SPLINE
SPL {X  -153.420, Y  +337.122, Z    +0.000, E1  +333.501, E3 -322809.091}
SPL {X  -157.288, Y  +353.220, Z    +0.000, E1  +341.134, E3 -322821.136}
SPL {X  -159.049, Y  +365.172, Z    +0.000, E1  +347.392, E3 -322826.689}
SPL {X  -159.749, Y  +373.719, Z    +0.000, E1  +352.250, E3 -322829.310}
SPL {X  -159.988, Y  +381.741, Z    +0.000, E1  +357.172, E3 -322830.785}
SPL {X  -159.990, Y  +387.352, Z    +0.000, E1  +361.387, E3 -322831.487}
SPL {X  -159.990, Y  +391.188, Z    +0.000, E1  +365.082, E3 -322832.027}
SPL {X  -159.990, Y  +395.106, Z    +0.000, E1  +369.154, E3 -322832.768}
SPL {X  -159.990, Y  +400.303, Z    +0.000, E1  +374.927, E3 -322834.090}
SPL {X  -159.990, Y  +408.423, Z    +0.000, E1  +383.302, E3 -322837.169}
SPL {X  -159.990, Y  +438.418, Z    +0.000, E1  +401.067, E3 -322858.742}
SPL {X  -159.990, Y  +482.913, Z    +0.000, E1  +407.036, E3 -322918.096}
SPL {X  -159.990, Y  +489.230, Z    +0.000, E1  +407.019, E3 -322930.608}
SPL {X  -159.990, Y  +495.241, Z    +0.000, E1  +407.026, E3 -322942.487}
SPL {X  -159.990, Y  +501.001, Z    +0.000, E1  +407.020, E3 -322953.864}
SPL {X  -159.990, Y  +506.758, Z    +0.000, E1  +407.038, E3 -322965.210}
SPL {X  -159.990, Y  +512.807, Z    +0.000, E1  +407.022, E3 -322977.201}
SPL {X  -159.990, Y  +518.043, Z    +0.000, E1  +407.016, E3 -322987.578}
SPL {X  -159.990, Y  +523.058, Z    +0.000, E1  +407.015, E3 -322997.494}
SPL {X  -159.990, Y  +527.746, Z    +0.000, E1  +407.012, E3 -323006.768}
SPL {X  -159.990, Y  +533.771, Z    +0.000, E1  +407.034, E3 -323018.653}
SPL {X  -159.990, Y  +542.379, Z    +0.000, E1  +407.067, E3 -323035.622}
SPL {X  -159.990, Y  +549.846, Z    +0.000, E1  +407.016, E3 -323050.468}
SPL {X  -159.990, Y  +554.843, Z    +0.000, E1  +407.014, E3 -323060.346}
SPL {X  -159.990, Y  +560.453, Z    +0.000, E1  +407.023, E3 -323071.429}
SPL {X  -159.990, Y  +566.612, Z    +0.000, E1  +407.022, E3 -323083.611}
SPL {X  -159.990, Y  +572.901, Z    +0.000, E1  +407.028, E3 -323096.022}
SPL {X  -159.990, Y  +578.640, Z    +0.000, E1  +407.021, E3 -323107.374}
SPL {X  -159.990, Y  +583.515, Z    +0.000, E1  +407.019, E3 -323117.014}
SPL {X  -159.990, Y  +589.675, Z    +0.000, E1  +407.042, E3 -323129.152}
SPL {X  -159.990, Y  +596.627, Z    +0.000, E1  +407.034, E3 -323142.892}
SPL {X  -159.990, Y  +602.039, Z    +0.000, E1  +407.021, E3 -323153.598}
SPL {X  -159.990, Y  +607.106, Z    +0.000, E1  +407.028, E3 -323163.605}
SPL {X  -159.990, Y  +612.418, Z    +0.000, E1  +407.023, E3 -323174.117}
SPL {X  -159.990, Y  +618.496, Z    +0.000, E1  +407.049, E3 -323186.084}
SPL {X  -159.990, Y  +624.357, Z    +0.000, E1  +407.020, E3 -323197.710}
SPL {X  -159.990, Y  +629.711, Z    +0.000, E1  +407.034, E3 -323208.279}
SPL {X  -159.990, Y  +635.041, Z    +0.000, E1  +407.022, E3 -323218.823}
SPL {X  -159.990, Y  +639.998, Z    +0.000, E1  +407.027, E3 -323228.616}
SPL {X  -159.990, Y  +646.188, Z    +0.000, E1  +407.041, E3 -323240.842}
SPL {X  -159.990, Y  +652.067, Z    +0.000, E1  +407.023, E3 -323252.478}
SPL {X  -159.990, Y  +657.109, Z    +0.000, E1  +407.025, E3 -323262.456}
SPL {X  -159.990, Y  +662.651, Z    +0.000, E1  +407.027, E3 -323273.412}
SPL {X  -159.990, Y  +668.015, Z    +0.000, E1  +407.025, E3 -323284.012}
SPL {X  -159.972, Y  +673.909, Z    +0.000, E1  +407.029, E3 -323295.678}
SPL {X  -159.776, Y  +679.772, Z    +0.000, E1  +406.992, E3 -323307.479}
SPL {X  -159.384, Y  +685.411, Z    +0.000, E1  +406.921, E3 -323319.040}
SPL {X  -158.839, Y  +690.657, Z    +0.000, E1  +406.819, E3 -323329.995}
SPL {X  -157.875, Y  +697.431, Z    +0.000, E1  +406.688, E3 -323344.334}
SPL {X  -156.719, Y  +703.686, Z    +0.000, E1  +406.438, E3 -323357.943}
SPL {X  -155.778, Y  +707.970, Z    +0.000, E1  +406.262, E3 -323367.418}
SPL {X  -154.419, Y  +713.351, Z    +0.000, E1  +406.025, E3 -323379.450}
SPL {X  -152.913, Y  +718.557, Z    +0.000, E1  +405.729, E3 -323391.301}
SPL {X  -151.262, Y  +723.621, Z    +0.000, E1  +405.429, E3 -323402.968}
SPL {X  -149.964, Y  +727.247, Z    +0.000, E1  +405.152, E3 -323411.472}
SPL {X  -148.611, Y  +730.759, Z    +0.000, E1  +404.909, E3 -323419.733}
SPL {X  -142.577, Y  +744.086, Z    +0.000, E1  +400.686, E3 -323483.103}
ENDSPLINE

SPLINE
SPL {X  -152.566, Y  +719.671, Z    +0.000, E1  +387.682, E3 -323553.573}
SPL {X  -158.253, Y  +695.011, Z    +0.000, E1  +375.913, E3 -323570.245}
SPL {X  -159.486, Y  +684.192, Z    +0.000, E1  +369.965, E3 -323574.192}
SPL {X  -159.898, Y  +676.924, Z    +0.000, E1  +365.683, E3 -323575.890}
SPL {X  -159.990, Y  +671.720, Z    +0.000, E1  +362.298, E3 -323576.730}
SPL {X  -159.990, Y  +668.164, Z    +0.000, E1  +359.695, E3 -323577.145}
SPL {X  -159.990, Y  +665.062, Z    +0.000, E1  +356.961, E3 -323577.485}
SPL {X  -159.990, Y  +660.795, Z    +0.000, E1  +352.651, E3 -323578.147}
SPL {X  -159.990, Y  +654.574, Z    +0.000, E1  +345.673, E3 -323579.602}
SPL {X  -159.990, Y  +647.816, Z    +0.000, E1  +338.252, E3 -323581.854}
SPL {X  -159.990, Y  +640.751, Z    +0.000, E1  +331.747, E3 -323585.447}
SPL {X  -159.990, Y  +611.706, Z    +0.000, E1  +317.244, E3 -323608.221}
SPL {X  -159.990, Y  +571.318, Z    +0.000, E1  +312.417, E3 -323661.605}
SPL {X  -159.990, Y  +564.395, Z    +0.000, E1  +312.373, E3 -323674.963}
SPL {X  -159.990, Y  +555.871, Z    +0.000, E1  +312.389, E3 -323691.511}
SPL {X  -159.990, Y  +549.223, Z    +0.000, E1  +312.413, E3 -323704.434}
SPL {X  -159.990, Y  +542.502, Z    +0.000, E1  +312.392, E3 -323717.432}
SPL {X  -159.990, Y  +536.986, Z    +0.000, E1  +312.423, E3 -323728.152}
SPL {X  -159.990, Y  +532.938, Z    +0.000, E1  +312.415, E3 -323735.979}
SPL {X  -159.990, Y  +527.222, Z    +0.000, E1  +312.401, E3 -323747.045}
SPL {X  -159.990, Y  +520.237, Z    +0.000, E1  +312.390, E3 -323760.575}
SPL {X  -159.990, Y  +514.002, Z    +0.000, E1  +312.418, E3 -323772.710}
SPL {X  -159.990, Y  +507.203, Z    +0.000, E1  +312.383, E3 -323785.836}
ENDSPLINE

SPLINE
SPL {X  -159.990, Y  +517.758, Z    +0.000, E1  +318.109, E3 -323796.409}
ENDSPLINE

SPLINE
SPL {X  -159.990, Y  +516.975, Z    +0.000, E1  +319.588, E3 -323807.472}
SPL {X  -159.990, Y  +508.583, Z    +0.000, E1  +318.552, E3 -323821.777}
SPL {X  -159.990, Y  +502.438, Z    +0.000, E1  +317.876, E3 -323832.280}
SPL {X  -159.990, Y  +494.810, Z    +0.000, E1  +316.979, E3 -323844.696}
SPL {X  -159.990, Y  +485.551, Z    +0.000, E1  +316.053, E3 -323859.885}
SPL {X  -159.990, Y  +477.585, Z    +0.000, E1  +315.156, E3 -323871.796}
SPL {X  -159.990, Y  +470.785, Z    +0.000, E1  +314.453, E3 -323881.968}
SPL {X  -159.990, Y  +463.371, Z    +0.000, E1  +313.690, E3 -323892.693}
SPL {X  -159.990, Y  +455.469, Z    +0.000, E1  +312.807, E3 -323903.219}
SPL {X  -159.990, Y  +445.848, Z    +0.000, E1  +311.866, E3 -323916.312}
SPL {X  -159.990, Y  +436.400, Z    +0.000, E1  +311.449, E3 -323931.693}
SPL {X  -159.990, Y  +429.614, Z    +0.000, E1  +311.486, E3 -323944.484}
SPL {X  -159.990, Y  +423.677, Z    +0.000, E1  +311.471, E3 -323955.595}
SPL {X  -159.990, Y  +417.714, Z    +0.000, E1  +311.484, E3 -323966.806}
SPL {X  -159.990, Y  +412.449, Z    +0.000, E1  +311.483, E3 -323976.666}
SPL {X  -159.990, Y  +406.256, Z    +0.000, E1  +311.459, E3 -323988.233}
SPL {X  -159.990, Y  +399.971, Z    +0.000, E1  +311.480, E3 -324000.048}
SPL {X  -159.990, Y  +394.711, Z    +0.000, E1  +311.476, E3 -324009.906}
SPL {X  -159.990, Y  +387.710, Z    +0.000, E1  +311.455, E3 -324023.029}
SPL {X  -159.966, Y  +379.751, Z    +0.000, E1  +311.465, E3 -324037.993}
SPL {X  -159.734, Y  +373.449, Z    +0.000, E1  +311.528, E3 -324050.097}
SPL {X  -159.358, Y  +368.299, Z    +0.000, E1  +311.595, E3 -324060.156}
SPL {X  -158.689, Y  +362.140, Z    +0.000, E1  +311.691, E3 -324072.383}
SPL {X  -157.692, Y  +355.479, Z    +0.000, E1  +311.882, E3 -324085.942}
SPL {X  -156.759, Y  +350.510, Z    +0.000, E1  +312.069, E3 -324096.257}
SPL {X  -155.408, Y  +344.485, Z    +0.000, E1  +312.267, E3 -324108.892}
SPL {X  -153.753, Y  +338.264, Z    +0.000, E1  +312.613, E3 -324122.322}
SPL {X  -152.142, Y  +333.005, Z    +0.000, E1  +312.891, E3 -324133.795}
SPL {X  -150.309, Y  +327.691, Z    +0.000, E1  +313.264, E3 -324145.650}
SPL {X  -148.834, Y  +323.804, Z    +0.000, E1  +313.556, E3 -324154.413}
SPL {X  -147.343, Y  +320.157, Z    +0.000, E1  +313.838, E3 -324162.703}
SPL {X  -142.380, Y  +309.529, Z    +0.000, E1  +319.953, E3 -324235.464}
ENDSPLINE

SPLINE
SPL {X  -153.420, Y  +337.122, Z    +0.000, E1  +333.501, E3 -324292.962}
SPL {X  -157.288, Y  +353.220, Z    +0.000, E1  +341.134, E3 -324305.007}
SPL {X  -159.049, Y  +365.172, Z    +0.000, E1  +347.392, E3 -324310.560}
SPL {X  -159.749, Y  +373.719, Z    +0.000, E1  +352.250, E3 -324313.181}
SPL {X  -159.988, Y  +381.741, Z    +0.000, E1  +357.172, E3 -324314.656}
SPL {X  -159.990, Y  +387.352, Z    +0.000, E1  +361.387, E3 -324315.358}
SPL {X  -159.990, Y  +392.444, Z    +0.000, E1  +366.277, E3 -324316.126}
SPL {X  -159.990, Y  +398.585, Z    +0.000, E1  +372.930, E3 -324317.506}
SPL {X  -159.990, Y  +408.423, Z    +0.000, E1  +383.302, E3 -324321.040}
SPL {X  -159.990, Y  +438.418, Z    +0.000, E1  +401.067, E3 -324342.613}
SPL {X  -159.990, Y  +482.913, Z    +0.000, E1  +407.036, E3 -324401.967}
SPL {X  -159.990, Y  +489.230, Z    +0.000, E1  +407.019, E3 -324414.479}
SPL {X  -159.990, Y  +495.241, Z    +0.000, E1  +407.026, E3 -324426.358}
SPL {X  -159.990, Y  +501.001, Z    +0.000, E1  +407.020, E3 -324437.735}
SPL {X  -159.990, Y  +506.758, Z    +0.000, E1  +407.038, E3 -324449.081}
SPL {X  -159.990, Y  +512.807, Z    +0.000, E1  +407.022, E3 -324461.072}
SPL {X  -159.990, Y  +518.043, Z    +0.000, E1  +407.016, E3 -324471.449}
SPL {X  -159.990, Y  +523.058, Z    +0.000, E1  +407.015, E3 -324481.365}
SPL {X  -159.990, Y  +527.746, Z    +0.000, E1  +407.012, E3 -324490.639}
SPL {X  -159.990, Y  +533.771, Z    +0.000, E1  +407.034, E3 -324502.523}
SPL {X  -159.990, Y  +542.379, Z    +0.000, E1  +407.067, E3 -324519.493}
SPL {X  -159.990, Y  +549.846, Z    +0.000, E1  +407.016, E3 -324534.339}
SPL {X  -159.990, Y  +554.843, Z    +0.000, E1  +407.014, E3 -324544.217}
SPL {X  -159.990, Y  +560.453, Z    +0.000, E1  +407.023, E3 -324555.299}
SPL {X  -159.990, Y  +566.612, Z    +0.000, E1  +407.022, E3 -324567.482}
SPL {X  -159.990, Y  +572.901, Z    +0.000, E1  +407.028, E3 -324579.893}
SPL {X  -159.990, Y  +578.640, Z    +0.000, E1  +407.021, E3 -324591.245}
SPL {X  -159.990, Y  +583.515, Z    +0.000, E1  +407.019, E3 -324600.885}
SPL {X  -159.990, Y  +589.675, Z    +0.000, E1  +407.042, E3 -324613.023}
SPL {X  -159.990, Y  +596.627, Z    +0.000, E1  +407.034, E3 -324626.763}
SPL {X  -159.990, Y  +602.039, Z    +0.000, E1  +407.021, E3 -324637.469}
SPL {X  -159.990, Y  +607.106, Z    +0.000, E1  +407.028, E3 -324647.476}
SPL {X  -159.990, Y  +614.483, Z    +0.000, E1  +407.064, E3 -324662.009}
SPL {X  -159.990, Y  +622.758, Z    +0.000, E1  +407.049, E3 -324678.379}
SPL {X  -159.990, Y  +629.711, Z    +0.000, E1  +407.034, E3 -324692.150}
SPL {X  -159.990, Y  +635.041, Z    +0.000, E1  +407.022, E3 -324702.694}
SPL {X  -159.990, Y  +639.998, Z    +0.000, E1  +407.027, E3 -324712.487}
SPL {X  -159.990, Y  +646.188, Z    +0.000, E1  +407.041, E3 -324724.713}
SPL {X  -159.990, Y  +652.067, Z    +0.000, E1  +407.023, E3 -324736.349}
SPL {X  -159.990, Y  +657.109, Z    +0.000, E1  +407.025, E3 -324746.327}
SPL {X  -159.990, Y  +662.651, Z    +0.000, E1  +407.027, E3 -324757.283}
SPL {X  -159.990, Y  +668.015, Z    +0.000, E1  +407.025, E3 -324767.883}
SPL {X  -159.972, Y  +673.909, Z    +0.000, E1  +407.029, E3 -324779.549}
SPL {X  -159.776, Y  +679.772, Z    +0.000, E1  +406.992, E3 -324791.350}
SPL {X  -159.384, Y  +685.411, Z    +0.000, E1  +406.921, E3 -324802.911}
SPL {X  -158.839, Y  +690.657, Z    +0.000, E1  +406.819, E3 -324813.865}
SPL {X  -157.875, Y  +697.431, Z    +0.000, E1  +406.688, E3 -324828.205}
SPL {X  -156.719, Y  +703.686, Z    +0.000, E1  +406.438, E3 -324841.814}
SPL {X  -155.432, Y  +709.417, Z    +0.000, E1  +406.234, E3 -324854.458}
SPL {X  -154.084, Y  +714.570, Z    +0.000, E1  +405.932, E3 -324866.120}
SPL {X  -152.913, Y  +718.557, Z    +0.000, E1  +405.729, E3 -324875.172}
SPL {X  -151.262, Y  +723.621, Z    +0.000, E1  +405.429, E3 -324886.839}
SPL {X  -149.074, Y  +729.584, Z    +0.000, E1  +405.040, E3 -324900.767}
SPL {X  -142.546, Y  +744.145, Z    +0.000, E1  +401.000, E3 -324963.794}
ENDSPLINE

SPLINE
SPL {X  -146.166, Y  +736.557, Z    +0.000, E1  +395.148, E3 -325007.760}
SPL {X  -153.596, Y  +716.277, Z    +0.000, E1  +386.138, E3 -325041.007}
SPL {X  -158.253, Y  +695.011, Z    +0.000, E1  +375.913, E3 -325054.116}
SPL {X  -159.486, Y  +684.192, Z    +0.000, E1  +369.965, E3 -325058.063}
SPL {X  -159.898, Y  +676.924, Z    +0.000, E1  +365.683, E3 -325059.761}
SPL {X  -159.990, Y  +671.720, Z    +0.000, E1  +362.298, E3 -325060.601}
SPL {X  -159.990, Y  +668.164, Z    +0.000, E1  +359.695, E3 -325061.016}
SPL {X  -159.990, Y  +663.705, Z    +0.000, E1  +355.772, E3 -325061.548}
SPL {X  -159.990, Y  +656.120, Z    +0.000, E1  +347.542, E3 -325063.089}
SPL {X  -159.990, Y  +647.816, Z    +0.000, E1  +338.252, E3 -325065.725}
SPL {X  -159.990, Y  +640.751, Z    +0.000, E1  +331.747, E3 -325069.318}
SPL {X  -159.990, Y  +611.706, Z    +0.000, E1  +317.244, E3 -325092.092}
SPL {X  -159.990, Y  +571.318, Z    +0.000, E1  +312.417, E3 -325145.476}
SPL {X  -159.990, Y  +564.395, Z    +0.000, E1  +312.373, E3 -325158.834}
SPL {X  -159.990, Y  +555.871, Z    +0.000, E1  +312.389, E3 -325175.382}
SPL {X  -159.990, Y  +549.223, Z    +0.000, E1  +312.413, E3 -325188.305}
SPL {X  -159.990, Y  +542.502, Z    +0.000, E1  +312.392, E3 -325201.303}
SPL {X  -159.990, Y  +536.986, Z    +0.000, E1  +312.423, E3 -325212.023}
SPL {X  -159.990, Y  +532.938, Z    +0.000, E1  +312.415, E3 -325219.850}
SPL {X  -159.990, Y  +527.222, Z    +0.000, E1  +312.401, E3 -325230.916}
SPL {X  -159.990, Y  +520.237, Z    +0.000, E1  +312.390, E3 -325244.446}
SPL {X  -159.990, Y  +514.002, Z    +0.000, E1  +312.418, E3 -325256.581}
SPL {X  -159.990, Y  +507.203, Z    +0.000, E1  +312.383, E3 -325269.707}
ENDSPLINE

SPLINE
SPL {X  -159.990, Y  +517.758, Z    +0.000, E1  +318.109, E3 -325280.280}
ENDSPLINE

SPLINE
SPL {X  -159.990, Y  +516.975, Z    +0.000, E1  +319.588, E3 -325291.343}
SPL {X  -159.990, Y  +508.583, Z    +0.000, E1  +318.552, E3 -325305.648}
SPL {X  -159.990, Y  +502.438, Z    +0.000, E1  +317.876, E3 -325316.151}
SPL {X  -159.990, Y  +494.810, Z    +0.000, E1  +316.979, E3 -325328.567}
SPL {X  -159.990, Y  +485.551, Z    +0.000, E1  +316.053, E3 -325343.756}
SPL {X  -159.990, Y  +477.585, Z    +0.000, E1  +315.156, E3 -325355.667}
SPL {X  -159.990, Y  +470.785, Z    +0.000, E1  +314.453, E3 -325365.839}
SPL {X  -159.990, Y  +463.371, Z    +0.000, E1  +313.690, E3 -325376.564}
SPL {X  -159.990, Y  +455.469, Z    +0.000, E1  +312.807, E3 -325387.090}
SPL {X  -159.990, Y  +445.848, Z    +0.000, E1  +311.866, E3 -325400.183}
SPL {X  -159.990, Y  +436.400, Z    +0.000, E1  +311.449, E3 -325415.564}
SPL {X  -159.990, Y  +429.614, Z    +0.000, E1  +311.486, E3 -325428.355}
SPL {X  -159.990, Y  +423.677, Z    +0.000, E1  +311.471, E3 -325439.466}
SPL {X  -159.990, Y  +417.714, Z    +0.000, E1  +311.484, E3 -325450.677}
SPL {X  -159.990, Y  +412.449, Z    +0.000, E1  +311.483, E3 -325460.537}
SPL {X  -159.990, Y  +406.256, Z    +0.000, E1  +311.459, E3 -325472.104}
SPL {X  -159.990, Y  +399.971, Z    +0.000, E1  +311.480, E3 -325483.919}
SPL {X  -159.990, Y  +392.623, Z    +0.000, E1  +311.440, E3 -325497.650}
SPL {X  -159.990, Y  +385.787, Z    +0.000, E1  +311.488, E3 -325510.557}
SPL {X  -159.966, Y  +379.751, Z    +0.000, E1  +311.465, E3 -325521.864}
SPL {X  -159.734, Y  +373.449, Z    +0.000, E1  +311.528, E3 -325533.968}
SPL {X  -159.230, Y  +366.920, Z    +0.000, E1  +311.592, E3 -325546.712}
SPL {X  -158.532, Y  +360.951, Z    +0.000, E1  +311.745, E3 -325558.686}
SPL {X  -157.692, Y  +355.479, Z    +0.000, E1  +311.882, E3 -325569.813}
SPL {X  -156.349, Y  +348.560, Z    +0.000, E1  +312.101, E3 -325584.153}
SPL {X  -154.984, Y  +342.790, Z    +0.000, E1  +312.392, E3 -325596.450}
SPL {X  -153.247, Y  +336.540, Z    +0.000, E1  +312.660, E3 -325609.885}
SPL {X  -150.765, Y  +328.959, Z    +0.000, E1  +313.136, E3 -325626.632}
SPL {X  -148.834, Y  +323.804, Z    +0.000, E1  +313.556, E3 -325638.284}
SPL {X  -147.343, Y  +320.157, Z    +0.000, E1  +313.838, E3 -325646.574}
SPL {X  -142.380, Y  +309.529, Z    +0.000, E1  +319.953, E3 -325719.335}
ENDSPLINE

SPLINE
SPL {X  -153.420, Y  +337.122, Z    +0.000, E1  +333.501, E3 -325776.833}
SPL {X  -157.288, Y  +353.220, Z    +0.000, E1  +341.134, E3 -325788.878}
SPL {X  -159.049, Y  +365.172, Z    +0.000, E1  +347.392, E3 -325794.431}
SPL {X  -159.749, Y  +373.719, Z    +0.000, E1  +352.250, E3 -325797.052}
SPL {X  -159.988, Y  +381.741, Z    +0.000, E1  +357.172, E3 -325798.527}
SPL {X  -159.990, Y  +387.352, Z    +0.000, E1  +361.387, E3 -325799.229}
SPL {X  -159.990, Y  +391.188, Z    +0.000, E1  +365.082, E3 -325799.769}
SPL {X  -159.990, Y  +395.106, Z    +0.000, E1  +369.154, E3 -325800.510}
SPL {X  -159.990, Y  +400.303, Z    +0.000, E1  +374.927, E3 -325801.832}
SPL {X  -159.990, Y  +408.423, Z    +0.000, E1  +383.302, E3 -325804.911}
SPL {X  -159.990, Y  +438.418, Z    +0.000, E1  +401.067, E3 -325826.484}
SPL {X  -159.990, Y  +482.913, Z    +0.000, E1  +407.036, E3 -325885.838}
SPL {X  -159.990, Y  +489.230, Z    +0.000, E1  +407.019, E3 -325898.350}
SPL {X  -159.990, Y  +495.241, Z    +0.000, E1  +407.026, E3 -325910.229}
SPL {X  -159.990, Y  +501.001, Z    +0.000, E1  +407.020, E3 -325921.606}
SPL {X  -159.990, Y  +506.758, Z    +0.000, E1  +407.038, E3 -325932.952}
SPL {X  -159.990, Y  +512.807, Z    +0.000, E1  +407.022, E3 -325944.943}
SPL {X  -159.990, Y  +518.043, Z    +0.000, E1  +407.016, E3 -325955.320}
SPL {X  -159.990, Y  +523.058, Z    +0.000, E1  +407.015, E3 -325965.236}
SPL {X  -159.990, Y  +527.746, Z    +0.000, E1  +407.012, E3 -325974.510}
SPL {X  -159.990, Y  +533.771, Z    +0.000, E1  +407.034, E3 -325986.394}
SPL {X  -159.990, Y  +542.379, Z    +0.000, E1  +407.067, E3 -326003.364}
SPL {X  -159.990, Y  +549.846, Z    +0.000, E1  +407.016, E3 -326018.210}
SPL {X  -159.990, Y  +554.843, Z    +0.000, E1  +407.014, E3 -326028.088}
SPL {X  -159.990, Y  +560.453, Z    +0.000, E1  +407.023, E3 -326039.170}
SPL {X  -159.990, Y  +566.612, Z    +0.000, E1  +407.022, E3 -326051.353}
SPL {X  -159.990, Y  +572.901, Z    +0.000, E1  +407.028, E3 -326063.764}
SPL {X  -159.990, Y  +578.640, Z    +0.000, E1  +407.021, E3 -326075.116}
SPL {X  -159.990, Y  +583.515, Z    +0.000, E1  +407.019, E3 -326084.756}
SPL {X  -159.990, Y  +589.675, Z    +0.000, E1  +407.042, E3 -326096.893}
SPL {X  -159.990, Y  +596.627, Z    +0.000, E1  +407.034, E3 -326110.634}
SPL {X  -159.990, Y  +602.039, Z    +0.000, E1  +407.021, E3 -326121.340}
SPL {X  -159.990, Y  +607.106, Z    +0.000, E1  +407.028, E3 -326131.347}
SPL {X  -159.990, Y  +612.418, Z    +0.000, E1  +407.023, E3 -326141.859}
SPL {X  -159.990, Y  +618.496, Z    +0.000, E1  +407.049, E3 -326153.826}
SPL {X  -159.990, Y  +624.357, Z    +0.000, E1  +407.020, E3 -326165.452}
SPL {X  -159.990, Y  +629.711, Z    +0.000, E1  +407.034, E3 -326176.021}
SPL {X  -159.990, Y  +635.041, Z    +0.000, E1  +407.022, E3 -326186.565}
SPL {X  -159.990, Y  +639.998, Z    +0.000, E1  +407.027, E3 -326196.358}
SPL {X  -159.990, Y  +646.188, Z    +0.000, E1  +407.041, E3 -326208.584}
SPL {X  -159.990, Y  +652.067, Z    +0.000, E1  +407.023, E3 -326220.220}
SPL {X  -159.990, Y  +657.109, Z    +0.000, E1  +407.025, E3 -326230.198}
SPL {X  -159.990, Y  +662.651, Z    +0.000, E1  +407.027, E3 -326241.154}
SPL {X  -159.990, Y  +668.015, Z    +0.000, E1  +407.025, E3 -326251.754}
SPL {X  -159.972, Y  +673.909, Z    +0.000, E1  +407.029, E3 -326263.420}
SPL {X  -159.776, Y  +679.772, Z    +0.000, E1  +406.992, E3 -326275.221}
SPL {X  -159.384, Y  +685.411, Z    +0.000, E1  +406.921, E3 -326286.782}
SPL {X  -158.839, Y  +690.657, Z    +0.000, E1  +406.819, E3 -326297.736}
SPL {X  -157.875, Y  +697.431, Z    +0.000, E1  +406.688, E3 -326312.076}
SPL {X  -156.719, Y  +703.686, Z    +0.000, E1  +406.438, E3 -326325.685}
SPL {X  -155.778, Y  +707.970, Z    +0.000, E1  +406.262, E3 -326335.160}
SPL {X  -154.419, Y  +713.351, Z    +0.000, E1  +406.025, E3 -326347.192}
SPL {X  -152.913, Y  +718.557, Z    +0.000, E1  +405.729, E3 -326359.043}
SPL {X  -151.262, Y  +723.621, Z    +0.000, E1  +405.429, E3 -326370.710}
SPL {X  -149.964, Y  +727.247, Z    +0.000, E1  +405.152, E3 -326379.214}
SPL {X  -148.611, Y  +730.759, Z    +0.000, E1  +404.909, E3 -326387.475}
SPL {X  -142.577, Y  +744.086, Z    +0.000, E1  +400.686, E3 -326450.844}
ENDSPLINE

SPLINE
SPL {X  -152.566, Y  +719.671, Z    +0.000, E1  +387.682, E3 -326521.315}
SPL {X  -158.253, Y  +695.011, Z    +0.000, E1  +375.913, E3 -326537.987}
SPL {X  -159.486, Y  +684.192, Z    +0.000, E1  +369.965, E3 -326541.934}
SPL {X  -159.898, Y  +676.924, Z    +0.000, E1  +365.683, E3 -326543.632}
SPL {X  -159.990, Y  +671.720, Z    +0.000, E1  +362.298, E3 -326544.472}
SPL {X  -159.990, Y  +668.164, Z    +0.000, E1  +359.695, E3 -326544.887}
SPL {X  -159.990, Y  +665.062, Z    +0.000, E1  +356.961, E3 -326545.227}
SPL {X  -159.990, Y  +660.795, Z    +0.000, E1  +352.651, E3 -326545.889}
SPL {X  -159.990, Y  +654.574, Z    +0.000, E1  +345.673, E3 -326547.344}
SPL {X  -159.990, Y  +647.816, Z    +0.000, E1  +338.252, E3 -326549.596}
SPL {X  -159.990, Y  +640.751, Z    +0.000, E1  +331.747, E3 -326553.189}
SPL {X  -159.990, Y  +611.706, Z    +0.000, E1  +317.244, E3 -326575.963}
SPL {X  -159.990, Y  +571.318, Z    +0.000, E1  +312.417, E3 -326629.347}
SPL {X  -159.990, Y  +564.395, Z    +0.000, E1  +312.373, E3 -326642.705}
SPL {X  -159.990, Y  +555.871, Z    +0.000, E1  +312.389, E3 -326659.253}
SPL {X  -159.990, Y  +549.223, Z    +0.000, E1  +312.413, E3 -326672.176}
SPL {X  -159.990, Y  +542.502, Z    +0.000, E1  +312.392, E3 -326685.174}
SPL {X  -159.990, Y  +536.986, Z    +0.000, E1  +312.423, E3 -326695.894}
SPL {X  -159.990, Y  +532.938, Z    +0.000, E1  +312.415, E3 -326703.721}
SPL {X  -159.990, Y  +527.222, Z    +0.000, E1  +312.401, E3 -326714.787}
SPL {X  -159.990, Y  +520.237, Z    +0.000, E1  +312.390, E3 -326728.317}
SPL {X  -159.990, Y  +514.002, Z    +0.000, E1  +312.418, E3 -326740.452}
SPL {X  -159.990, Y  +507.203, Z    +0.000, E1  +312.383, E3 -326753.578}
ENDSPLINE

SPLINE
SPL {X  -159.990, Y  +517.758, Z    +0.000, E1  +318.109, E3 -326764.151}
ENDSPLINE

SPLINE
SPL {X  -159.990, Y  +516.975, Z    +0.000, E1  +319.588, E3 -326775.214}
SPL {X  -159.990, Y  +508.583, Z    +0.000, E1  +318.552, E3 -326789.519}
SPL {X  -159.990, Y  +502.438, Z    +0.000, E1  +317.876, E3 -326800.022}
SPL {X  -159.990, Y  +494.810, Z    +0.000, E1  +316.979, E3 -326812.438}
SPL {X  -159.990, Y  +485.551, Z    +0.000, E1  +316.053, E3 -326827.627}
SPL {X  -159.990, Y  +477.585, Z    +0.000, E1  +315.156, E3 -326839.538}
SPL {X  -159.990, Y  +470.785, Z    +0.000, E1  +314.453, E3 -326849.710}
SPL {X  -159.990, Y  +463.371, Z    +0.000, E1  +313.690, E3 -326860.435}
SPL {X  -159.990, Y  +455.469, Z    +0.000, E1  +312.807, E3 -326870.961}
SPL {X  -159.990, Y  +445.848, Z    +0.000, E1  +311.866, E3 -326884.054}
SPL {X  -159.990, Y  +436.400, Z    +0.000, E1  +311.449, E3 -326899.435}
SPL {X  -159.990, Y  +429.614, Z    +0.000, E1  +311.486, E3 -326912.226}
SPL {X  -159.990, Y  +423.677, Z    +0.000, E1  +311.471, E3 -326923.337}
SPL {X  -159.990, Y  +417.714, Z    +0.000, E1  +311.484, E3 -326934.547}
SPL {X  -159.990, Y  +412.449, Z    +0.000, E1  +311.483, E3 -326944.408}
SPL {X  -159.990, Y  +406.256, Z    +0.000, E1  +311.459, E3 -326955.975}
SPL {X  -159.990, Y  +399.971, Z    +0.000, E1  +311.480, E3 -326967.790}
SPL {X  -159.990, Y  +394.711, Z    +0.000, E1  +311.476, E3 -326977.648}
SPL {X  -159.990, Y  +387.710, Z    +0.000, E1  +311.455, E3 -326990.771}
SPL {X  -159.966, Y  +379.751, Z    +0.000, E1  +311.465, E3 -327005.735}
SPL {X  -159.734, Y  +373.449, Z    +0.000, E1  +311.528, E3 -327017.839}
SPL {X  -159.358, Y  +368.299, Z    +0.000, E1  +311.595, E3 -327027.898}
SPL {X  -158.689, Y  +362.140, Z    +0.000, E1  +311.691, E3 -327040.125}
SPL {X  -157.692, Y  +355.479, Z    +0.000, E1  +311.882, E3 -327053.684}
SPL {X  -156.759, Y  +350.510, Z    +0.000, E1  +312.069, E3 -327063.999}
SPL {X  -155.408, Y  +344.485, Z    +0.000, E1  +312.267, E3 -327076.634}
SPL {X  -153.753, Y  +338.264, Z    +0.000, E1  +312.613, E3 -327090.064}
SPL {X  -152.142, Y  +333.005, Z    +0.000, E1  +312.891, E3 -327101.537}
SPL {X  -150.309, Y  +327.691, Z    +0.000, E1  +313.264, E3 -327113.392}
SPL {X  -148.834, Y  +323.804, Z    +0.000, E1  +313.556, E3 -327122.155}
SPL {X  -147.343, Y  +320.157, Z    +0.000, E1  +313.838, E3 -327130.445}
SPL {X  -142.380, Y  +309.529, Z    +0.000, E1  +319.953, E3 -327203.206}
ENDSPLINE

SPLINE
SPL {X  -153.420, Y  +337.122, Z    +0.000, E1  +333.501, E3 -327260.704}
SPL {X  -157.288, Y  +353.220, Z    +0.000, E1  +341.134, E3 -327272.749}
SPL {X  -159.049, Y  +365.172, Z    +0.000, E1  +347.392, E3 -327278.302}
SPL {X  -159.749, Y  +373.719, Z    +0.000, E1  +352.250, E3 -327280.923}
SPL {X  -159.988, Y  +381.741, Z    +0.000, E1  +357.172, E3 -327282.398}
SPL {X  -159.990, Y  +387.352, Z    +0.000, E1  +361.387, E3 -327283.100}
SPL {X  -159.990, Y  +392.444, Z    +0.000, E1  +366.277, E3 -327283.868}
SPL {X  -159.990, Y  +398.585, Z    +0.000, E1  +372.930, E3 -327285.248}
SPL {X  -159.990, Y  +408.423, Z    +0.000, E1  +383.302, E3 -327288.782}
SPL {X  -159.990, Y  +438.418, Z    +0.000, E1  +401.067, E3 -327310.355}
SPL {X  -159.990, Y  +482.913, Z    +0.000, E1  +407.036, E3 -327369.709}
SPL {X  -159.990, Y  +489.230, Z    +0.000, E1  +407.019, E3 -327382.221}
SPL {X  -159.990, Y  +495.241, Z    +0.000, E1  +407.026, E3 -327394.100}
SPL {X  -159.990, Y  +501.001, Z    +0.000, E1  +407.020, E3 -327405.477}
SPL {X  -159.990, Y  +506.758, Z    +0.000, E1  +407.038, E3 -327416.823}
SPL {X  -159.990, Y  +512.807, Z    +0.000, E1  +407.022, E3 -327428.814}
SPL {X  -159.990, Y  +518.043, Z    +0.000, E1  +407.016, E3 -327439.191}
SPL {X  -159.990, Y  +525.485, Z    +0.000, E1  +407.063, E3 -327453.836}
SPL {X  -159.990, Y  +533.771, Z    +0.000, E1  +407.034, E3 -327470.265}
SPL {X  -159.990, Y  +540.264, Z    +0.000, E1  +407.020, E3 -327483.122}
SPL {X  -159.990, Y  +547.787, Z    +0.000, E1  +407.067, E3 -327497.923}
SPL {X  -159.990, Y  +554.843, Z    +0.000, E1  +407.014, E3 -327511.959}
SPL {X  -159.990, Y  +560.453, Z    +0.000, E1  +407.023, E3 -327523.041}
SPL {X  -159.990, Y  +566.612, Z    +0.000, E1  +407.022, E3 -327535.224}
SPL {X  -159.990, Y  +572.901, Z    +0.000, E1  +407.028, E3 -327547.635}
SPL {X  -159.990, Y  +578.640, Z    +0.000, E1  +407.021, E3 -327558.987}
SPL {X  -159.990, Y  +584.969, Z    +0.000, E1  +407.043, E3 -327571.469}
SPL {X  -159.990, Y  +591.074, Z    +0.000, E1  +407.017, E3 -327583.559}
SPL {X  -159.990, Y  +596.627, Z    +0.000, E1  +407.034, E3 -327594.505}
SPL {X  -159.990, Y  +602.039, Z    +0.000, E1  +407.021, E3 -327605.211}
SPL {X  -159.990, Y  +607.106, Z    +0.000, E1  +407.028, E3 -327615.218}
SPL {X  -159.990, Y  +612.418, Z    +0.000, E1  +407.023, E3 -327625.730}
SPL {X  -159.990, Y  +618.496, Z    +0.000, E1  +407.049, E3 -327637.697}
SPL {X  -159.990, Y  +624.357, Z    +0.000, E1  +407.020, E3 -327649.323}
SPL {X  -159.990, Y  +629.711, Z    +0.000, E1  +407.034, E3 -327659.892}
SPL {X  -159.990, Y  +635.041, Z    +0.000, E1  +407.022, E3 -327670.436}
SPL {X  -159.990, Y  +642.261, Z    +0.000, E1  +407.074, E3 -327684.637}
SPL {X  -159.990, Y  +650.752, Z    +0.000, E1  +407.046, E3 -327701.464}
SPL {X  -159.990, Y  +657.109, Z    +0.000, E1  +407.025, E3 -327714.069}
SPL {X  -159.990, Y  +662.651, Z    +0.000, E1  +407.027, E3 -327725.025}
SPL {X  -159.990, Y  +668.015, Z    +0.000, E1  +407.025, E3 -327735.625}
SPL {X  -159.972, Y  +673.909, Z    +0.000, E1  +407.029, E3 -327747.291}
SPL {X  -159.776, Y  +679.772, Z    +0.000, E1  +406.992, E3 -327759.092}
SPL {X  -159.384, Y  +685.411, Z    +0.000, E1  +406.921, E3 -327770.653}
SPL {X  -158.642, Y  +692.228, Z    +0.000, E1  +406.819, E3 -327784.869}
SPL {X  -157.651, Y  +698.760, Z    +0.000, E1  +406.609, E3 -327798.863}
SPL {X  -156.719, Y  +703.686, Z    +0.000, E1  +406.438, E3 -327809.556}
SPL {X  -155.778, Y  +707.970, Z    +0.000, E1  +406.262, E3 -327819.031}
SPL {X  -154.419, Y  +713.351, Z    +0.000, E1  +406.025, E3 -327831.062}
SPL {X  -152.913, Y  +718.557, Z    +0.000, E1  +405.729, E3 -327842.914}
SPL {X  -151.262, Y  +723.621, Z    +0.000, E1  +405.429, E3 -327854.581}
SPL {X  -149.074, Y  +729.584, Z    +0.000, E1  +405.040, E3 -327868.509}
SPL {X  -142.577, Y  +744.086, Z    +0.000, E1  +400.686, E3 -327934.715}
ENDSPLINE

SPLINE
SPL {X  -152.566, Y  +719.671, Z    +0.000, E1  +387.682, E3 -328005.186}
SPL {X  -158.253, Y  +695.011, Z    +0.000, E1  +375.913, E3 -328021.858}
SPL {X  -159.486, Y  +684.192, Z    +0.000, E1  +369.965, E3 -328025.805}
SPL {X  -159.898, Y  +676.924, Z    +0.000, E1  +365.683, E3 -328027.503}
SPL {X  -159.990, Y  +671.720, Z    +0.000, E1  +362.298, E3 -328028.343}
SPL {X  -159.990, Y  +668.164, Z    +0.000, E1  +359.695, E3 -328028.758}
SPL {X  -159.990, Y  +665.062, Z    +0.000, E1  +356.961, E3 -328029.098}
SPL {X  -159.990, Y  +660.795, Z    +0.000, E1  +352.651, E3 -328029.760}
SPL {X  -159.990, Y  +654.574, Z    +0.000, E1  +345.673, E3 -328031.215}
SPL {X  -159.990, Y  +644.002, Z    +0.000, E1  +334.724, E3 -328035.412}
SPL {X  -159.990, Y  +611.706, Z    +0.000, E1  +317.244, E3 -328059.834}
SPL {X  -159.990, Y  +571.318, Z    +0.000, E1  +312.417, E3 -328113.218}
SPL {X  -159.990, Y  +564.395, Z    +0.000, E1  +312.373, E3 -328126.576}
SPL {X  -159.990, Y  +555.871, Z    +0.000, E1  +312.389, E3 -328143.124}
SPL {X  -159.990, Y  +549.223, Z    +0.000, E1  +312.413, E3 -328156.047}
SPL {X  -159.990, Y  +542.502, Z    +0.000, E1  +312.392, E3 -328169.045}
SPL {X  -159.990, Y  +534.538, Z    +0.000, E1  +312.385, E3 -328184.449}
SPL {X  -159.990, Y  +527.222, Z    +0.000, E1  +312.401, E3 -328198.658}
SPL {X  -159.990, Y  +520.237, Z    +0.000, E1  +312.390, E3 -328212.188}
SPL {X  -159.990, Y  +512.328, Z    +0.000, E1  +312.388, E3 -328227.522}
SPL {X  -159.990, Y  +505.755, Z    +0.000, E1  +312.413, E3 -328240.299}
ENDSPLINE

SPLINE
SPL {X  -159.990, Y  +518.404, Z    +0.000, E1  +319.229, E3 -328253.546}
ENDSPLINE

SPLINE
SPL {X  -159.990, Y  +509.980, Z    +0.000, E1  +318.692, E3 -328270.950}
SPL {X  -159.990, Y  +499.983, Z    +0.000, E1  +317.561, E3 -328287.845}
SPL {X  -159.990, Y  +490.062, Z    +0.000, E1  +316.490, E3 -328304.128}
SPL {X  -159.990, Y  +479.678, Z    +0.000, E1  +315.383, E3 -328320.348}
SPL {X  -159.990, Y  +470.785, Z    +0.000, E1  +314.453, E3 -328333.581}
SPL {X  -159.990, Y  +463.371, Z    +0.000, E1  +313.690, E3 -328344.306}
SPL {X  -159.990, Y  +453.200, Z    +0.000, E1  +312.569, E3 -328357.946}
SPL {X  -159.990, Y  +441.904, Z    +0.000, E1  +311.574, E3 -328373.659}
SPL {X  -159.990, Y  +434.881, Z    +0.000, E1  +311.481, E3 -328386.208}
SPL {X  -159.990, Y  +427.340, Z    +0.000, E1  +311.445, E3 -328400.301}
SPL {X  -159.990, Y  +418.926, Z    +0.000, E1  +311.461, E3 -328416.110}
SPL {X  -159.990, Y  +412.449, Z    +0.000, E1  +311.483, E3 -328428.279}
SPL {X  -159.990, Y  +406.256, Z    +0.000, E1  +311.459, E3 -328439.846}
SPL {X  -159.990, Y  +399.971, Z    +0.000, E1  +311.480, E3 -328451.661}
SPL {X  -159.990, Y  +392.623, Z    +0.000, E1  +311.440, E3 -328465.392}
SPL {X  -159.990, Y  +383.159, Z    +0.000, E1  +311.442, E3 -328483.161}
SPL {X  -159.797, Y  +374.648, Z    +0.000, E1  +311.491, E3 -328499.354}
SPL {X  -159.358, Y  +368.299, Z    +0.000, E1  +311.595, E3 -328511.769}
SPL {X  -158.689, Y  +362.140, Z    +0.000, E1  +311.691, E3 -328523.996}
SPL {X  -157.692, Y  +355.479, Z    +0.000, E1  +311.882, E3 -328537.555}
SPL {X  -156.349, Y  +348.560, Z    +0.000, E1  +312.101, E3 -328551.895}
SPL {X  -154.984, Y  +342.790, Z    +0.000, E1  +312.392, E3 -328564.192}
SPL {X  -153.247, Y  +336.540, Z    +0.000, E1  +312.660, E3 -328577.627}
SPL {X  -150.765, Y  +328.959, Z    +0.000, E1  +313.136, E3 -328594.374}
SPL {X  -148.834, Y  +323.804, Z    +0.000, E1  +313.556, E3 -328606.026}
SPL {X  -147.343, Y  +320.157, Z    +0.000, E1  +313.838, E3 -328614.316}
SPL {X  -142.380, Y  +309.529, Z    +0.000, E1  +319.953, E3 -328687.077}
ENDSPLINE

SPLINE
SPL {X  -153.420, Y  +337.122, Z    +0.000, E1  +333.501, E3 -328744.575}
SPL {X  -157.288, Y  +353.220, Z    +0.000, E1  +341.134, E3 -328756.620}
SPL {X  -159.049, Y  +365.172, Z    +0.000, E1  +347.392, E3 -328762.173}
SPL {X  -159.881, Y  +376.607, Z    +0.000, E1  +353.914, E3 -328765.402}
SPL {X  -159.990, Y  +383.110, Z    +0.000, E1  +358.202, E3 -328766.455}
SPL {X  -159.990, Y  +387.352, Z    +0.000, E1  +361.387, E3 -328766.971}
SPL {X  -159.990, Y  +391.188, Z    +0.000, E1  +365.082, E3 -328767.511}
SPL {X  -159.990, Y  +395.106, Z    +0.000, E1  +369.154, E3 -328768.252}
SPL {X  -159.990, Y  +400.303, Z    +0.000, E1  +374.927, E3 -328769.574}
SPL {X  -159.990, Y  +408.423, Z    +0.000, E1  +383.302, E3 -328772.653}
SPL {X  -159.990, Y  +438.418, Z    +0.000, E1  +401.067, E3 -328794.226}
SPL {X  -159.990, Y  +482.913, Z    +0.000, E1  +407.036, E3 -328853.580}
SPL {X  -159.990, Y  +489.230, Z    +0.000, E1  +407.019, E3 -328866.092}
SPL {X  -159.990, Y  +495.241, Z    +0.000, E1  +407.026, E3 -328877.971}
SPL {X  -159.990, Y  +501.001, Z    +0.000, E1  +407.020, E3 -328889.347}
SPL {X  -159.990, Y  +506.758, Z    +0.000, E1  +407.038, E3 -328900.694}
SPL {X  -159.990, Y  +512.807, Z    +0.000, E1  +407.022, E3 -328912.685}
SPL {X  -159.990, Y  +518.043, Z    +0.000, E1  +407.016, E3 -328923.062}
SPL {X  -159.990, Y  +523.058, Z    +0.000, E1  +407.015, E3 -328932.978}
SPL {X  -159.990, Y  +527.746, Z    +0.000, E1  +407.012, E3 -328942.252}
SPL {X  -159.990, Y  +533.771, Z    +0.000, E1  +407.034, E3 -328954.136}
SPL {X  -159.990, Y  +542.379, Z    +0.000, E1  +407.067, E3 -328971.106}
SPL {X  -159.990, Y  +549.846, Z    +0.000, E1  +407.016, E3 -328985.952}
SPL {X  -159.990, Y  +554.843, Z    +0.000, E1  +407.014, E3 -328995.830}
SPL {X  -159.990, Y  +560.453, Z    +0.000, E1  +407.023, E3 -329006.912}
SPL {X  -159.990, Y  +566.612, Z    +0.000, E1  +407.022, E3 -329019.095}
SPL {X  -159.990, Y  +572.901, Z    +0.000, E1  +407.028, E3 -329031.506}
SPL {X  -159.990, Y  +578.640, Z    +0.000, E1  +407.021, E3 -329042.858}
SPL {X  -159.990, Y  +583.515, Z    +0.000, E1  +407.019, E3 -329052.498}
SPL {X  -159.990, Y  +589.675, Z    +0.000, E1  +407.042, E3 -329064.635}
SPL {X  -159.990, Y  +596.627, Z    +0.000, E1  +407.034, E3 -329078.375}
SPL {X  -159.990, Y  +602.039, Z    +0.000, E1  +407.021, E3 -329089.082}
SPL {X  -159.990, Y  +607.106, Z    +0.000, E1  +407.028, E3 -329099.089}
SPL {X  -159.990, Y  +612.418, Z    +0.000, E1  +407.023, E3 -329109.601}
SPL {X  -159.990, Y  +618.496, Z    +0.000, E1  +407.049, E3 -329121.568}
SPL {X  -159.990, Y  +624.357, Z    +0.000, E1  +407.020, E3 -329133.194}
SPL {X  -159.990, Y  +629.711, Z    +0.000, E1  +407.034, E3 -329143.763}
SPL {X  -159.990, Y  +635.041, Z    +0.000, E1  +407.022, E3 -329154.307}
SPL {X  -159.990, Y  +639.998, Z    +0.000, E1  +407.027, E3 -329164.100}
SPL {X  -159.990, Y  +646.188, Z    +0.000, E1  +407.041, E3 -329176.326}
SPL {X  -159.990, Y  +652.067, Z    +0.000, E1  +407.023, E3 -329187.962}
SPL {X  -159.990, Y  +657.109, Z    +0.000, E1  +407.025, E3 -329197.940}
SPL {X  -159.990, Y  +662.651, Z    +0.000, E1  +407.027, E3 -329208.896}
SPL {X  -159.990, Y  +668.015, Z    +0.000, E1  +407.025, E3 -329219.496}
SPL {X  -159.972, Y  +673.909, Z    +0.000, E1  +407.029, E3 -329231.162}
SPL {X  -159.776, Y  +679.772, Z    +0.000, E1  +406.992, E3 -329242.963}
SPL {X  -159.384, Y  +685.411, Z    +0.000, E1  +406.921, E3 -329254.524}
SPL {X  -158.642, Y  +692.228, Z    +0.000, E1  +406.819, E3 -329268.740}
SPL {X  -157.651, Y  +698.760, Z    +0.000, E1  +406.609, E3 -329282.734}
SPL {X  -156.719, Y  +703.686, Z    +0.000, E1  +406.438, E3 -329293.427}
SPL {X  -155.778, Y  +707.970, Z    +0.000, E1  +406.262, E3 -329302.902}
SPL {X  -154.419, Y  +713.351, Z    +0.000, E1  +406.025, E3 -329314.933}
SPL {X  -152.913, Y  +718.557, Z    +0.000, E1  +405.729, E3 -329326.785}
SPL {X  -151.262, Y  +723.621, Z    +0.000, E1  +405.429, E3 -329338.452}
SPL {X  -149.074, Y  +729.584, Z    +0.000, E1  +405.040, E3 -329352.380}
SPL {X  -142.577, Y  +744.086, Z    +0.000, E1  +400.686, E3 -329418.586}
ENDSPLINE

SPLINE
SPL {X  -152.566, Y  +719.671, Z    +0.000, E1  +387.682, E3 -329489.057}
SPL {X  -158.253, Y  +695.011, Z    +0.000, E1  +375.913, E3 -329505.729}
SPL {X  -159.486, Y  +684.192, Z    +0.000, E1  +369.965, E3 -329509.676}
SPL {X  -159.898, Y  +676.924, Z    +0.000, E1  +365.683, E3 -329511.374}
SPL {X  -159.990, Y  +671.720, Z    +0.000, E1  +362.298, E3 -329512.214}
SPL {X  -159.990, Y  +668.164, Z    +0.000, E1  +359.695, E3 -329512.629}
SPL {X  -159.990, Y  +665.062, Z    +0.000, E1  +356.961, E3 -329512.969}
SPL {X  -159.990, Y  +660.795, Z    +0.000, E1  +352.651, E3 -329513.631}
SPL {X  -159.990, Y  +654.574, Z    +0.000, E1  +345.673, E3 -329515.086}
SPL {X  -159.990, Y  +647.816, Z    +0.000, E1  +338.252, E3 -329517.338}
SPL {X  -159.990, Y  +640.751, Z    +0.000, E1  +331.747, E3 -329520.931}
SPL {X  -159.990, Y  +611.706, Z    +0.000, E1  +317.244, E3 -329543.705}
SPL {X  -159.990, Y  +567.814, Z    +0.000, E1  +312.360, E3 -329603.794}
SPL {X  -159.990, Y  +558.774, Z    +0.000, E1  +312.384, E3 -329621.360}
SPL {X  -159.990, Y  +550.551, Z    +0.000, E1  +312.385, E3 -329637.301}
SPL {X  -159.990, Y  +542.502, Z    +0.000, E1  +312.392, E3 -329652.916}
SPL {X  -159.990, Y  +536.986, Z    +0.000, E1  +312.423, E3 -329663.636}
SPL {X  -159.990, Y  +532.938, Z    +0.000, E1  +312.415, E3 -329671.463}
SPL {X  -159.990, Y  +525.893, Z    +0.000, E1  +312.375, E3 -329685.076}
SPL {X  -159.990, Y  +518.864, Z    +0.000, E1  +312.415, E3 -329698.759}
SPL {X  -159.990, Y  +512.328, Z    +0.000, E1  +312.388, E3 -329711.393}
SPL {X  -159.990, Y  +505.755, Z    +0.000, E1  +312.413, E3 -329724.170}
ENDSPLINE

SPLINE
SPL {X  -159.990, Y  +517.758, Z    +0.000, E1  +318.109, E3 -329731.893}
ENDSPLINE

SPLINE
SPL {X  -159.990, Y  +516.975, Z    +0.000, E1  +319.588, E3 -329742.956}
SPL {X  -159.990, Y  +508.583, Z    +0.000, E1  +318.552, E3 -329757.261}
SPL {X  -159.990, Y  +499.983, Z    +0.000, E1  +317.561, E3 -329771.716}
SPL {X  -159.990, Y  +492.624, Z    +0.000, E1  +316.776, E3 -329783.819}
SPL {X  -159.990, Y  +485.551, Z    +0.000, E1  +316.053, E3 -329795.369}
SPL {X  -159.990, Y  +477.585, Z    +0.000, E1  +315.156, E3 -329807.280}
SPL {X  -159.990, Y  +470.785, Z    +0.000, E1  +314.453, E3 -329817.452}
SPL {X  -159.990, Y  +463.371, Z    +0.000, E1  +313.690, E3 -329828.177}
SPL {X  -159.990, Y  +455.469, Z    +0.000, E1  +312.807, E3 -329838.703}
SPL {X  -159.990, Y  +445.848, Z    +0.000, E1  +311.866, E3 -329851.796}
SPL {X  -159.990, Y  +436.400, Z    +0.000, E1  +311.449, E3 -329867.177}
SPL {X  -159.990, Y  +429.614, Z    +0.000, E1  +311.486, E3 -329879.967}
SPL {X  -159.990, Y  +423.677, Z    +0.000, E1  +311.471, E3 -329891.079}
SPL {X  -159.990, Y  +417.714, Z    +0.000, E1  +311.484, E3 -329902.289}
SPL {X  -159.990, Y  +412.449, Z    +0.000, E1  +311.483, E3 -329912.150}
SPL {X  -159.990, Y  +406.256, Z    +0.000, E1  +311.459, E3 -329923.717}
SPL {X  -159.990, Y  +399.971, Z    +0.000, E1  +311.480, E3 -329935.532}
SPL {X  -159.990, Y  +394.711, Z    +0.000, E1  +311.476, E3 -329945.390}
SPL {X  -159.990, Y  +387.710, Z    +0.000, E1  +311.455, E3 -329958.513}
SPL {X  -159.966, Y  +379.751, Z    +0.000, E1  +311.465, E3 -329973.477}
SPL {X  -159.734, Y  +373.449, Z    +0.000, E1  +311.528, E3 -329985.581}
SPL {X  -159.230, Y  +366.920, Z    +0.000, E1  +311.592, E3 -329998.325}
SPL {X  -158.532, Y  +360.951, Z    +0.000, E1  +311.745, E3 -330010.299}
SPL {X  -157.692, Y  +355.479, Z    +0.000, E1  +311.882, E3 -330021.426}
SPL {X  -156.349, Y  +348.560, Z    +0.000, E1  +312.101, E3 -330035.766}
SPL {X  -154.984, Y  +342.790, Z    +0.000, E1  +312.392, E3 -330048.063}
SPL {X  -153.247, Y  +336.540, Z    +0.000, E1  +312.660, E3 -330061.498}
SPL {X  -150.765, Y  +328.959, Z    +0.000, E1  +313.136, E3 -330078.245}
SPL {X  -148.834, Y  +323.804, Z    +0.000, E1  +313.556, E3 -330089.897}
SPL {X  -147.343, Y  +320.157, Z    +0.000, E1  +313.838, E3 -330098.187}
SPL {X  -142.380, Y  +309.529, Z    +0.000, E1  +319.953, E3 -330170.948}
ENDSPLINE

SPLINE
SPL {X  -153.420, Y  +337.122, Z    +0.000, E1  +333.501, E3 -330228.446}
SPL {X  -157.288, Y  +353.220, Z    +0.000, E1  +341.134, E3 -330240.491}
SPL {X  -159.049, Y  +365.172, Z    +0.000, E1  +347.392, E3 -330246.044}
SPL {X  -159.749, Y  +373.719, Z    +0.000, E1  +352.250, E3 -330248.665}
SPL {X  -159.988, Y  +381.741, Z    +0.000, E1  +357.172, E3 -330250.140}
SPL {X  -159.990, Y  +387.352, Z    +0.000, E1  +361.387, E3 -330250.842}
SPL {X  -159.990, Y  +391.188, Z    +0.000, E1  +365.082, E3 -330251.382}
SPL {X  -159.990, Y  +395.106, Z    +0.000, E1  +369.154, E3 -330252.123}
SPL {X  -159.990, Y  +400.303, Z    +0.000, E1  +374.927, E3 -330253.445}
SPL {X  -159.990, Y  +408.423, Z    +0.000, E1  +383.302, E3 -330256.524}
SPL {X  -159.990, Y  +438.418, Z    +0.000, E1  +401.067, E3 -330278.097}
SPL {X  -159.990, Y  +482.913, Z    +0.000, E1  +407.036, E3 -330337.451}
SPL {X  -159.990, Y  +489.230, Z    +0.000, E1  +407.019, E3 -330349.963}
SPL {X  -159.990, Y  +495.241, Z    +0.000, E1  +407.026, E3 -330361.842}
SPL {X  -159.990, Y  +501.001, Z    +0.000, E1  +407.020, E3 -330373.218}
SPL {X  -159.990, Y  +506.758, Z    +0.000, E1  +407.038, E3 -330384.565}
SPL {X  -159.990, Y  +512.807, Z    +0.000, E1  +407.022, E3 -330396.556}
SPL {X  -159.990, Y  +518.043, Z    +0.000, E1  +407.016, E3 -330406.933}
SPL {X  -159.990, Y  +523.058, Z    +0.000, E1  +407.015, E3 -330416.849}
SPL {X  -159.990, Y  +527.746, Z    +0.000, E1  +407.012, E3 -330426.123}
SPL {X  -159.990, Y  +533.771, Z    +0.000, E1  +407.034, E3 -330438.007}
SPL {X  -159.990, Y  +542.379, Z    +0.000, E1  +407.067, E3 -330454.977}
SPL {X  -159.990, Y  +549.846, Z    +0.000, E1  +407.016, E3 -330469.822}
SPL {X  -159.990, Y  +554.843, Z    +0.000, E1  +407.014, E3 -330479.701}
SPL {X  -159.990, Y  +560.453, Z    +0.000, E1  +407.023, E3 -330490.783}
SPL {X  -159.990, Y  +566.612, Z    +0.000, E1  +407.022, E3 -330502.966}
SPL {X  -159.990, Y  +572.901, Z    +0.000, E1  +407.028, E3 -330515.377}
SPL {X  -159.990, Y  +578.640, Z    +0.000, E1  +407.021, E3 -330526.729}
SPL {X  -159.990, Y  +584.969, Z    +0.000, E1  +407.043, E3 -330539.211}
SPL {X  -159.990, Y  +591.074, Z    +0.000, E1  +407.017, E3 -330551.301}
SPL {X  -159.990, Y  +596.627, Z    +0.000, E1  +407.034, E3 -330562.246}
SPL {X  -159.990, Y  +602.039, Z    +0.000, E1  +407.021, E3 -330572.953}
SPL {X  -159.990, Y  +607.106, Z    +0.000, E1  +407.028, E3 -330582.960}
SPL {X  -159.990, Y  +612.418, Z    +0.000, E1  +407.023, E3 -330593.472}
SPL {X  -159.990, Y  +618.496, Z    +0.000, E1  +407.049, E3 -330605.439}
SPL {X  -159.990, Y  +624.357, Z    +0.000, E1  +407.020, E3 -330617.065}
SPL {X  -159.990, Y  +629.711, Z    +0.000, E1  +407.034, E3 -330627.634}
SPL {X  -159.990, Y  +635.041, Z    +0.000, E1  +407.022, E3 -330638.178}
SPL {X  -159.990, Y  +639.998, Z    +0.000, E1  +407.027, E3 -330647.970}
SPL {X  -159.990, Y  +646.188, Z    +0.000, E1  +407.041, E3 -330660.197}
SPL {X  -159.990, Y  +652.067, Z    +0.000, E1  +407.023, E3 -330671.832}
SPL {X  -159.990, Y  +657.109, Z    +0.000, E1  +407.025, E3 -330681.811}
SPL {X  -159.990, Y  +662.651, Z    +0.000, E1  +407.027, E3 -330692.767}
SPL {X  -159.990, Y  +668.015, Z    +0.000, E1  +407.025, E3 -330703.367}
SPL {X  -159.972, Y  +673.909, Z    +0.000, E1  +407.029, E3 -330715.033}
SPL {X  -159.776, Y  +679.772, Z    +0.000, E1  +406.992, E3 -330726.834}
SPL {X  -159.384, Y  +685.411, Z    +0.000, E1  +406.921, E3 -330738.395}
SPL {X  -158.642, Y  +692.228, Z    +0.000, E1  +406.819, E3 -330752.611}
SPL {X  -157.651, Y  +698.760, Z    +0.000, E1  +406.609, E3 -330766.605}
SPL {X  -156.719, Y  +703.686, Z    +0.000, E1  +406.438, E3 -330777.298}
SPL {X  -155.778, Y  +707.970, Z    +0.000, E1  +406.262, E3 -330786.773}
SPL {X  -154.419, Y  +713.351, Z    +0.000, E1  +406.025, E3 -330798.804}
SPL {X  -152.913, Y  +718.557, Z    +0.000, E1  +405.729, E3 -330810.656}
SPL {X  -151.262, Y  +723.621, Z    +0.000, E1  +405.429, E3 -330822.323}
SPL {X  -149.074, Y  +729.584, Z    +0.000, E1  +405.040, E3 -330836.251}
SPL {X  -142.577, Y  +744.086, Z    +0.000, E1  +400.686, E3 -330902.457}
ENDSPLINE

SPLINE
SPL {X  -152.566, Y  +719.671, Z    +0.000, E1  +387.682, E3 -330972.928}
SPL {X  -158.253, Y  +695.011, Z    +0.000, E1  +375.913, E3 -330989.600}
SPL {X  -159.486, Y  +684.192, Z    +0.000, E1  +369.965, E3 -330993.547}
SPL {X  -159.898, Y  +676.924, Z    +0.000, E1  +365.683, E3 -330995.245}
SPL {X  -159.990, Y  +671.720, Z    +0.000, E1  +362.298, E3 -330996.085}
SPL {X  -159.990, Y  +668.164, Z    +0.000, E1  +359.695, E3 -330996.500}
SPL {X  -159.990, Y  +665.062, Z    +0.000, E1  +356.961, E3 -330996.840}
SPL {X  -159.990, Y  +660.795, Z    +0.000, E1  +352.651, E3 -330997.502}
SPL {X  -159.990, Y  +654.574, Z    +0.000, E1  +345.673, E3 -330998.957}
SPL {X  -159.990, Y  +644.002, Z    +0.000, E1  +334.724, E3 -331003.154}
SPL {X  -159.990, Y  +611.706, Z    +0.000, E1  +317.244, E3 -331027.576}
SPL {X  -159.990, Y  +571.318, Z    +0.000, E1  +312.417, E3 -331080.960}
SPL {X  -159.990, Y  +566.024, Z    +0.000, E1  +312.406, E3 -331091.209}
SPL {X  -159.990, Y  +558.774, Z    +0.000, E1  +312.384, E3 -331105.231}
SPL {X  -159.990, Y  +550.551, Z    +0.000, E1  +312.385, E3 -331121.172}
SPL {X  -159.990, Y  +542.502, Z    +0.000, E1  +312.392, E3 -331136.787}
SPL {X  -159.990, Y  +534.538, Z    +0.000, E1  +312.385, E3 -331152.191}
SPL {X  -159.990, Y  +527.222, Z    +0.000, E1  +312.401, E3 -331166.399}
SPL {X  -159.990, Y  +520.237, Z    +0.000, E1  +312.390, E3 -331179.930}
SPL {X  -159.990, Y  +512.328, Z    +0.000, E1  +312.388, E3 -331195.264}
SPL {X  -159.990, Y  +505.755, Z    +0.000, E1  +312.413, E3 -331208.041}
ENDSPLINE

SPLINE
SPL {X  -159.990, Y  +517.758, Z    +0.000, E1  +318.109, E3 -331215.763}
ENDSPLINE

SPLINE
SPL {X  -159.990, Y  +516.975, Z    +0.000, E1  +319.588, E3 -331226.827}
SPL {X  -159.990, Y  +508.583, Z    +0.000, E1  +318.552, E3 -331241.132}
SPL {X  -159.990, Y  +502.438, Z    +0.000, E1  +317.876, E3 -331251.635}
SPL {X  -159.990, Y  +494.810, Z    +0.000, E1  +316.979, E3 -331264.051}
SPL {X  -159.990, Y  +487.314, Z    +0.000, E1  +316.246, E3 -331276.419}
SPL {X  -159.990, Y  +479.678, Z    +0.000, E1  +315.383, E3 -331288.090}
SPL {X  -159.990, Y  +470.785, Z    +0.000, E1  +314.453, E3 -331301.323}
SPL {X  -159.990, Y  +463.371, Z    +0.000, E1  +313.690, E3 -331312.048}
SPL {X  -159.990, Y  +455.469, Z    +0.000, E1  +312.807, E3 -331322.574}
SPL {X  -159.990, Y  +449.689, Z    +0.000, E1  +312.264, E3 -331330.564}
SPL {X  -159.990, Y  +441.904, Z    +0.000, E1  +311.574, E3 -331341.401}
SPL {X  -159.990, Y  +434.881, Z    +0.000, E1  +311.481, E3 -331353.950}
SPL {X  -159.990, Y  +427.340, Z    +0.000, E1  +311.445, E3 -331368.043}
SPL {X  -159.990, Y  +418.926, Z    +0.000, E1  +311.461, E3 -331383.852}
SPL {X  -159.990, Y  +412.449, Z    +0.000, E1  +311.483, E3 -331396.021}
SPL {X  -159.990, Y  +406.256, Z    +0.000, E1  +311.459, E3 -331407.588}
SPL {X  -159.990, Y  +399.971, Z    +0.000, E1  +311.480, E3 -331419.403}
SPL {X  -159.990, Y  +392.623, Z    +0.000, E1  +311.440, E3 -331433.134}
SPL {X  -159.990, Y  +385.787, Z    +0.000, E1  +311.488, E3 -331446.041}
SPL {X  -159.966, Y  +379.751, Z    +0.000, E1  +311.465, E3 -331457.348}
SPL {X  -159.734, Y  +373.449, Z    +0.000, E1  +311.528, E3 -331469.452}
SPL {X  -159.230, Y  +366.920, Z    +0.000, E1  +311.592, E3 -331482.196}
SPL {X  -158.532, Y  +360.951, Z    +0.000, E1  +311.745, E3 -331494.170}
SPL {X  -157.692, Y  +355.479, Z    +0.000, E1  +311.882, E3 -331505.297}
SPL {X  -156.349, Y  +348.560, Z    +0.000, E1  +312.101, E3 -331519.636}
SPL {X  -154.984, Y  +342.790, Z    +0.000, E1  +312.392, E3 -331531.934}
SPL {X  -153.247, Y  +336.540, Z    +0.000, E1  +312.660, E3 -331545.369}
SPL {X  -150.765, Y  +328.959, Z    +0.000, E1  +313.136, E3 -331562.116}
SPL {X  -148.834, Y  +323.804, Z    +0.000, E1  +313.556, E3 -331573.768}
SPL {X  -147.343, Y  +320.157, Z    +0.000, E1  +313.838, E3 -331582.058}
SPL {X  -142.380, Y  +309.529, Z    +0.000, E1  +319.953, E3 -331654.819}
ENDSPLINE

SPLINE
SPL {X  -153.420, Y  +337.122, Z    +0.000, E1  +333.501, E3 -331712.317}
SPL {X  -157.288, Y  +353.220, Z    +0.000, E1  +341.134, E3 -331724.362}
SPL {X  -159.049, Y  +365.172, Z    +0.000, E1  +347.392, E3 -331729.915}
SPL {X  -159.881, Y  +376.607, Z    +0.000, E1  +353.914, E3 -331733.144}
SPL {X  -159.990, Y  +384.736, Z    +0.000, E1  +359.276, E3 -331734.395}
SPL {X  -159.990, Y  +389.821, Z    +0.000, E1  +363.632, E3 -331735.048}
SPL {X  -159.990, Y  +395.106, Z    +0.000, E1  +369.154, E3 -331735.994}
SPL {X  -159.990, Y  +400.303, Z    +0.000, E1  +374.927, E3 -331737.316}
SPL {X  -159.990, Y  +408.423, Z    +0.000, E1  +383.302, E3 -331740.395}
SPL {X  -159.990, Y  +438.418, Z    +0.000, E1  +401.067, E3 -331761.967}
SPL {X  -159.990, Y  +482.913, Z    +0.000, E1  +407.036, E3 -331821.322}
SPL {X  -159.990, Y  +489.230, Z    +0.000, E1  +407.019, E3 -331833.834}
SPL {X  -159.990, Y  +495.241, Z    +0.000, E1  +407.026, E3 -331845.713}
SPL {X  -159.990, Y  +501.001, Z    +0.000, E1  +407.020, E3 -331857.089}
SPL {X  -159.990, Y  +506.758, Z    +0.000, E1  +407.038, E3 -331868.436}
SPL {X  -159.990, Y  +512.807, Z    +0.000, E1  +407.022, E3 -331880.427}
SPL {X  -159.990, Y  +518.043, Z    +0.000, E1  +407.016, E3 -331890.804}
SPL {X  -159.990, Y  +523.058, Z    +0.000, E1  +407.015, E3 -331900.720}
SPL {X  -159.990, Y  +527.746, Z    +0.000, E1  +407.012, E3 -331909.994}
SPL {X  -159.990, Y  +533.771, Z    +0.000, E1  +407.034, E3 -331921.878}
SPL {X  -159.990, Y  +542.379, Z    +0.000, E1  +407.067, E3 -331938.848}
SPL {X  -159.990, Y  +549.846, Z    +0.000, E1  +407.016, E3 -331953.693}
SPL {X  -159.990, Y  +554.843, Z    +0.000, E1  +407.014, E3 -331963.572}
SPL {X  -159.990, Y  +560.453, Z    +0.000, E1  +407.023, E3 -331974.654}
SPL {X  -159.990, Y  +566.612, Z    +0.000, E1  +407.022, E3 -331986.837}
SPL {X  -159.990, Y  +572.901, Z    +0.000, E1  +407.028, E3 -331999.248}
SPL {X  -159.990, Y  +578.640, Z    +0.000, E1  +407.021, E3 -332010.600}
SPL {X  -159.990, Y  +583.515, Z    +0.000, E1  +407.019, E3 -332020.239}
SPL {X  -159.990, Y  +589.675, Z    +0.000, E1  +407.042, E3 -332032.377}
SPL {X  -159.990, Y  +596.627, Z    +0.000, E1  +407.034, E3 -332046.117}
SPL {X  -159.990, Y  +602.039, Z    +0.000, E1  +407.021, E3 -332056.824}
SPL {X  -159.990, Y  +607.106, Z    +0.000, E1  +407.028, E3 -332066.831}
SPL {X  -159.990, Y  +612.418, Z    +0.000, E1  +407.023, E3 -332077.343}
SPL {X  -159.990, Y  +618.496, Z    +0.000, E1  +407.049, E3 -332089.310}
SPL {X  -159.990, Y  +624.357, Z    +0.000, E1  +407.020, E3 -332100.936}
SPL {X  -159.990, Y  +629.711, Z    +0.000, E1  +407.034, E3 -332111.505}
SPL {X  -159.990, Y  +635.041, Z    +0.000, E1  +407.022, E3 -332122.049}
SPL {X  -159.990, Y  +639.998, Z    +0.000, E1  +407.027, E3 -332131.841}
SPL {X  -159.990, Y  +646.188, Z    +0.000, E1  +407.041, E3 -332144.068}
SPL {X  -159.990, Y  +652.067, Z    +0.000, E1  +407.023, E3 -332155.703}
SPL {X  -159.990, Y  +657.109, Z    +0.000, E1  +407.025, E3 -332165.682}
SPL {X  -159.990, Y  +662.651, Z    +0.000, E1  +407.027, E3 -332176.638}
SPL {X  -159.990, Y  +668.015, Z    +0.000, E1  +407.025, E3 -332187.238}
SPL {X  -159.972, Y  +673.909, Z    +0.000, E1  +407.029, E3 -332198.904}
SPL {X  -159.776, Y  +679.772, Z    +0.000, E1  +406.992, E3 -332210.705}
SPL {X  -159.384, Y  +685.411, Z    +0.000, E1  +406.921, E3 -332222.266}
SPL {X  -158.642, Y  +692.228, Z    +0.000, E1  +406.819, E3 -332236.482}
SPL {X  -157.651, Y  +698.760, Z    +0.000, E1  +406.609, E3 -332250.476}
SPL {X  -156.719, Y  +703.686, Z    +0.000, E1  +406.438, E3 -332261.169}
SPL {X  -155.778, Y  +707.970, Z    +0.000, E1  +406.262, E3 -332270.644}
SPL {X  -154.419, Y  +713.351, Z    +0.000, E1  +406.025, E3 -332282.675}
SPL {X  -152.913, Y  +718.557, Z    +0.000, E1  +405.729, E3 -332294.527}
SPL {X  -151.262, Y  +723.621, Z    +0.000, E1  +405.429, E3 -332306.194}
SPL {X  -149.074, Y  +729.584, Z    +0.000, E1  +405.040, E3 -332320.122}
SPL {X  -142.577, Y  +744.086, Z    +0.000, E1  +400.686, E3 -332386.328}
ENDSPLINE

SPLINE
SPL {X  -152.566, Y  +719.671, Z    +0.000, E1  +387.682, E3 -332456.799}
SPL {X  -158.253, Y  +695.011, Z    +0.000, E1  +375.913, E3 -332473.471}
SPL {X  -159.486, Y  +684.192, Z    +0.000, E1  +369.965, E3 -332477.418}
SPL {X  -159.898, Y  +676.924, Z    +0.000, E1  +365.683, E3 -332479.116}
SPL {X  -159.990, Y  +671.720, Z    +0.000, E1  +362.298, E3 -332479.956}
SPL {X  -159.990, Y  +668.164, Z    +0.000, E1  +359.695, E3 -332480.371}
SPL {X  -159.990, Y  +665.062, Z    +0.000, E1  +356.961, E3 -332480.711}
SPL {X  -159.990, Y  +660.795, Z    +0.000, E1  +352.651, E3 -332481.373}
SPL {X  -159.990, Y  +654.574, Z    +0.000, E1  +345.673, E3 -332482.828}
SPL {X  -159.990, Y  +647.816, Z    +0.000, E1  +338.252, E3 -332485.080}
SPL {X  -159.990, Y  +640.751, Z    +0.000, E1  +331.747, E3 -332488.673}
SPL {X  -159.990, Y  +611.706, Z    +0.000, E1  +317.244, E3 -332511.447}
SPL {X  -159.990, Y  +567.814, Z    +0.000, E1  +312.360, E3 -332571.536}
SPL {X  -159.990, Y  +558.774, Z    +0.000, E1  +312.384, E3 -332589.102}
SPL {X  -159.990, Y  +550.551, Z    +0.000, E1  +312.385, E3 -332605.043}
SPL {X  -159.990, Y  +542.502, Z    +0.000, E1  +312.392, E3 -332620.658}
SPL {X  -159.990, Y  +536.986, Z    +0.000, E1  +312.423, E3 -332631.378}
SPL {X  -159.990, Y  +532.938, Z    +0.000, E1  +312.415, E3 -332639.205}
SPL {X  -159.990, Y  +525.893, Z    +0.000, E1  +312.375, E3 -332652.818}
SPL {X  -159.990, Y  +518.864, Z    +0.000, E1  +312.415, E3 -332666.501}
SPL {X  -159.990, Y  +512.328, Z    +0.000, E1  +312.388, E3 -332679.135}
SPL {X  -159.990, Y  +505.755, Z    +0.000, E1  +312.413, E3 -332691.912}
ENDSPLINE

SPLINE
SPL {X  -159.990, Y  +517.758, Z    +0.000, E1  +318.109, E3 -332699.634}
ENDSPLINE

SPLINE
SPL {X  -159.990, Y  +516.975, Z    +0.000, E1  +319.588, E3 -332710.698}
SPL {X  -159.990, Y  +508.583, Z    +0.000, E1  +318.552, E3 -332725.003}
SPL {X  -159.990, Y  +499.983, Z    +0.000, E1  +317.561, E3 -332739.458}
SPL {X  -159.990, Y  +492.624, Z    +0.000, E1  +316.776, E3 -332751.561}
SPL {X  -159.990, Y  +485.551, Z    +0.000, E1  +316.053, E3 -332763.111}
SPL {X  -159.990, Y  +477.585, Z    +0.000, E1  +315.156, E3 -332775.022}
SPL {X  -159.990, Y  +470.785, Z    +0.000, E1  +314.453, E3 -332785.194}
SPL {X  -159.990, Y  +463.371, Z    +0.000, E1  +313.690, E3 -332795.919}
SPL {X  -159.990, Y  +455.469, Z    +0.000, E1  +312.807, E3 -332806.445}
SPL {X  -159.990, Y  +445.848, Z    +0.000, E1  +311.866, E3 -332819.538}
SPL {X  -159.990, Y  +436.400, Z    +0.000, E1  +311.449, E3 -332834.919}
SPL {X  -159.990, Y  +429.614, Z    +0.000, E1  +311.486, E3 -332847.709}
SPL {X  -159.990, Y  +423.677, Z    +0.000, E1  +311.471, E3 -332858.821}
SPL {X  -159.990, Y  +417.714, Z    +0.000, E1  +311.484, E3 -332870.031}
SPL {X  -159.990, Y  +412.449, Z    +0.000, E1  +311.483, E3 -332879.892}
SPL {X  -159.990, Y  +406.256, Z    +0.000, E1  +311.459, E3 -332891.459}
SPL {X  -159.990, Y  +399.971, Z    +0.000, E1  +311.480, E3 -332903.274}
SPL {X  -159.990, Y  +394.711, Z    +0.000, E1  +311.476, E3 -332913.132}
SPL {X  -159.990, Y  +387.710, Z    +0.000, E1  +311.455, E3 -332926.255}
SPL {X  -159.966, Y  +379.751, Z    +0.000, E1  +311.465, E3 -332941.219}
SPL {X  -159.734, Y  +373.449, Z    +0.000, E1  +311.528, E3 -332953.323}
SPL {X  -159.230, Y  +366.920, Z    +0.000, E1  +311.592, E3 -332966.067}
SPL {X  -158.532, Y  +360.951, Z    +0.000, E1  +311.745, E3 -332978.040}
SPL {X  -157.692, Y  +355.479, Z    +0.000, E1  +311.882, E3 -332989.168}
SPL {X  -156.349, Y  +348.560, Z    +0.000, E1  +312.101, E3 -333003.507}
SPL {X  -154.984, Y  +342.790, Z    +0.000, E1  +312.392, E3 -333015.805}
SPL {X  -153.247, Y  +336.540, Z    +0.000, E1  +312.660, E3 -333029.240}
SPL {X  -150.765, Y  +328.959, Z    +0.000, E1  +313.136, E3 -333045.987}
SPL {X  -148.834, Y  +323.804, Z    +0.000, E1  +313.556, E3 -333057.639}
SPL {X  -147.343, Y  +320.157, Z    +0.000, E1  +313.838, E3 -333065.929}
SPL {X  -142.380, Y  +309.529, Z    +0.000, E1  +319.953, E3 -333138.690}
ENDSPLINE

SPLINE
SPL {X  -153.420, Y  +337.122, Z    +0.000, E1  +333.501, E3 -333196.187}
SPL {X  -157.288, Y  +353.220, Z    +0.000, E1  +341.134, E3 -333208.233}
SPL {X  -159.049, Y  +365.172, Z    +0.000, E1  +347.392, E3 -333213.786}
SPL {X  -159.749, Y  +373.719, Z    +0.000, E1  +352.250, E3 -333216.407}
SPL {X  -159.988, Y  +381.741, Z    +0.000, E1  +357.172, E3 -333217.882}
SPL {X  -159.990, Y  +387.352, Z    +0.000, E1  +361.387, E3 -333218.584}
SPL {X  -159.990, Y  +391.188, Z    +0.000, E1  +365.082, E3 -333219.124}
SPL {X  -159.990, Y  +395.106, Z    +0.000, E1  +369.154, E3 -333219.865}
SPL {X  -159.990, Y  +400.303, Z    +0.000, E1  +374.927, E3 -333221.187}
SPL {X  -159.990, Y  +408.423, Z    +0.000, E1  +383.302, E3 -333224.266}
SPL {X  -159.990, Y  +438.418, Z    +0.000, E1  +401.067, E3 -333245.838}
SPL {X  -159.990, Y  +482.913, Z    +0.000, E1  +407.036, E3 -333305.193}
SPL {X  -159.990, Y  +489.230, Z    +0.000, E1  +407.019, E3 -333317.704}
SPL {X  -159.990, Y  +495.241, Z    +0.000, E1  +407.026, E3 -333329.584}
SPL {X  -159.990, Y  +501.001, Z    +0.000, E1  +407.020, E3 -333340.960}
SPL {X  -159.990, Y  +506.758, Z    +0.000, E1  +407.038, E3 -333352.306}
SPL {X  -159.990, Y  +512.807, Z    +0.000, E1  +407.022, E3 -333364.298}
SPL {X  -159.990, Y  +518.043, Z    +0.000, E1  +407.016, E3 -333374.675}
SPL {X  -159.990, Y  +523.058, Z    +0.000, E1  +407.015, E3 -333384.591}
SPL {X  -159.990, Y  +527.746, Z    +0.000, E1  +407.012, E3 -333393.865}
SPL {X  -159.990, Y  +533.771, Z    +0.000, E1  +407.034, E3 -333405.749}
SPL {X  -159.990, Y  +542.379, Z    +0.000, E1  +407.067, E3 -333422.719}
SPL {X  -159.990, Y  +549.846, Z    +0.000, E1  +407.016, E3 -333437.564}
SPL {X  -159.990, Y  +554.843, Z    +0.000, E1  +407.014, E3 -333447.443}
SPL {X  -159.990, Y  +560.453, Z    +0.000, E1  +407.023, E3 -333458.525}
SPL {X  -159.990, Y  +566.612, Z    +0.000, E1  +407.022, E3 -333470.708}
SPL {X  -159.990, Y  +572.901, Z    +0.000, E1  +407.028, E3 -333483.119}
SPL {X  -159.990, Y  +578.640, Z    +0.000, E1  +407.021, E3 -333494.471}
SPL {X  -159.990, Y  +584.969, Z    +0.000, E1  +407.043, E3 -333506.953}
SPL {X  -159.990, Y  +591.074, Z    +0.000, E1  +407.017, E3 -333519.043}
SPL {X  -159.990, Y  +596.627, Z    +0.000, E1  +407.034, E3 -333529.988}
SPL {X  -159.990, Y  +602.039, Z    +0.000, E1  +407.021, E3 -333540.695}
SPL {X  -159.990, Y  +607.106, Z    +0.000, E1  +407.028, E3 -333550.702}
SPL {X  -159.990, Y  +612.418, Z    +0.000, E1  +407.023, E3 -333561.214}
SPL {X  -159.990, Y  +618.496, Z    +0.000, E1  +407.049, E3 -333573.180}
SPL {X  -159.990, Y  +624.357, Z    +0.000, E1  +407.020, E3 -333584.806}
SPL {X  -159.990, Y  +629.711, Z    +0.000, E1  +407.034, E3 -333595.376}
SPL {X  -159.990, Y  +635.041, Z    +0.000, E1  +407.022, E3 -333605.920}
SPL {X  -159.990, Y  +639.998, Z    +0.000, E1  +407.027, E3 -333615.712}
SPL {X  -159.990, Y  +646.188, Z    +0.000, E1  +407.041, E3 -333627.939}
SPL {X  -159.990, Y  +652.067, Z    +0.000, E1  +407.023, E3 -333639.574}
SPL {X  -159.990, Y  +657.109, Z    +0.000, E1  +407.025, E3 -333649.553}
SPL {X  -159.990, Y  +662.651, Z    +0.000, E1  +407.027, E3 -333660.509}
SPL {X  -159.990, Y  +668.015, Z    +0.000, E1  +407.025, E3 -333671.109}
SPL {X  -159.972, Y  +673.909, Z    +0.000, E1  +407.029, E3 -333682.775}
SPL {X  -159.776, Y  +679.772, Z    +0.000, E1  +406.992, E3 -333694.576}
SPL {X  -159.384, Y  +685.411, Z    +0.000, E1  +406.921, E3 -333706.137}
SPL {X  -158.642, Y  +692.228, Z    +0.000, E1  +406.819, E3 -333720.353}
SPL {X  -157.651, Y  +698.760, Z    +0.000, E1  +406.609, E3 -333734.347}
SPL {X  -156.719, Y  +703.686, Z    +0.000, E1  +406.438, E3 -333745.040}
SPL {X  -155.778, Y  +707.970, Z    +0.000, E1  +406.262, E3 -333754.515}
SPL {X  -154.419, Y  +713.351, Z    +0.000, E1  +406.025, E3 -333766.546}
SPL {X  -152.913, Y  +718.557, Z    +0.000, E1  +405.729, E3 -333778.398}
SPL {X  -151.262, Y  +723.621, Z    +0.000, E1  +405.429, E3 -333790.065}
SPL {X  -149.074, Y  +729.584, Z    +0.000, E1  +405.040, E3 -333803.993}
SPL {X  -142.577, Y  +744.086, Z    +0.000, E1  +400.686, E3 -333870.199}
ENDSPLINE

SPLINE
SPL {X  -152.566, Y  +719.671, Z    +0.000, E1  +387.682, E3 -333940.670}
SPL {X  -158.253, Y  +695.011, Z    +0.000, E1  +375.913, E3 -333957.342}
SPL {X  -159.486, Y  +684.192, Z    +0.000, E1  +369.965, E3 -333961.289}
SPL {X  -159.898, Y  +676.924, Z    +0.000, E1  +365.683, E3 -333962.987}
SPL {X  -159.990, Y  +671.720, Z    +0.000, E1  +362.298, E3 -333963.827}
SPL {X  -159.990, Y  +668.164, Z    +0.000, E1  +359.695, E3 -333964.242}
SPL {X  -159.990, Y  +665.062, Z    +0.000, E1  +356.961, E3 -333964.582}
SPL {X  -159.990, Y  +660.795, Z    +0.000, E1  +352.651, E3 -333965.244}
SPL {X  -159.990, Y  +654.574, Z    +0.000, E1  +345.673, E3 -333966.699}
SPL {X  -159.990, Y  +644.002, Z    +0.000, E1  +334.724, E3 -333970.896}
SPL {X  -159.990, Y  +611.706, Z    +0.000, E1  +317.244, E3 -333995.318}
SPL {X  -159.990, Y  +571.318, Z    +0.000, E1  +312.417, E3 -334048.701}
SPL {X  -159.990, Y  +566.024, Z    +0.000, E1  +312.406, E3 -334058.951}
SPL {X  -159.990, Y  +558.774, Z    +0.000, E1  +312.384, E3 -334072.973}
SPL {X  -159.990, Y  +550.551, Z    +0.000, E1  +312.385, E3 -334088.914}
SPL {X  -159.990, Y  +542.502, Z    +0.000, E1  +312.392, E3 -334104.529}
SPL {X  -159.990, Y  +534.538, Z    +0.000, E1  +312.385, E3 -334119.933}
SPL {X  -159.990, Y  +527.222, Z    +0.000, E1  +312.401, E3 -334134.141}
SPL {X  -159.990, Y  +520.237, Z    +0.000, E1  +312.390, E3 -334147.672}
SPL {X  -159.990, Y  +512.328, Z    +0.000, E1  +312.388, E3 -334163.006}
SPL {X  -159.990, Y  +505.755, Z    +0.000, E1  +312.413, E3 -334175.783}
ENDSPLINE

SPLINE
SPL {X  -159.990, Y  +517.758, Z    +0.000, E1  +318.109, E3 -334183.505}
ENDSPLINE

SPLINE
SPL {X  -159.990, Y  +516.975, Z    +0.000, E1  +319.588, E3 -334194.569}
SPL {X  -159.990, Y  +508.583, Z    +0.000, E1  +318.552, E3 -334208.874}
SPL {X  -159.990, Y  +502.438, Z    +0.000, E1  +317.876, E3 -334219.377}
SPL {X  -159.990, Y  +494.810, Z    +0.000, E1  +316.979, E3 -334231.793}
SPL {X  -159.990, Y  +487.314, Z    +0.000, E1  +316.246, E3 -334244.161}
SPL {X  -159.990, Y  +479.678, Z    +0.000, E1  +315.383, E3 -334255.832}
SPL {X  -159.990, Y  +470.785, Z    +0.000, E1  +314.453, E3 -334269.065}
SPL {X  -159.990, Y  +463.371, Z    +0.000, E1  +313.690, E3 -334279.790}
SPL {X  -159.990, Y  +455.469, Z    +0.000, E1  +312.807, E3 -334290.316}
SPL {X  -159.990, Y  +449.689, Z    +0.000, E1  +312.264, E3 -334298.306}
SPL {X  -159.990, Y  +441.904, Z    +0.000, E1  +311.574, E3 -334309.143}
SPL {X  -159.990, Y  +434.881, Z    +0.000, E1  +311.481, E3 -334321.692}
SPL {X  -159.990, Y  +427.340, Z    +0.000, E1  +311.445, E3 -334335.785}
SPL {X  -159.990, Y  +418.926, Z    +0.000, E1  +311.461, E3 -334351.594}
SPL {X  -159.990, Y  +412.449, Z    +0.000, E1  +311.483, E3 -334363.763}
SPL {X  -159.990, Y  +406.256, Z    +0.000, E1  +311.459, E3 -334375.330}
SPL {X  -159.990, Y  +399.971, Z    +0.000, E1  +311.480, E3 -334387.145}
SPL {X  -159.990, Y  +392.623, Z    +0.000, E1  +311.440, E3 -334400.876}
SPL {X  -159.990, Y  +385.787, Z    +0.000, E1  +311.488, E3 -334413.783}
SPL {X  -159.966, Y  +379.751, Z    +0.000, E1  +311.465, E3 -334425.090}
SPL {X  -159.734, Y  +373.449, Z    +0.000, E1  +311.528, E3 -334437.194}
SPL {X  -159.230, Y  +366.920, Z    +0.000, E1  +311.592, E3 -334449.938}
SPL {X  -158.532, Y  +360.951, Z    +0.000, E1  +311.745, E3 -334461.911}
SPL {X  -157.692, Y  +355.479, Z    +0.000, E1  +311.882, E3 -334473.039}
SPL {X  -156.349, Y  +348.560, Z    +0.000, E1  +312.101, E3 -334487.378}
SPL {X  -154.984, Y  +342.790, Z    +0.000, E1  +312.392, E3 -334499.676}
SPL {X  -153.247, Y  +336.540, Z    +0.000, E1  +312.660, E3 -334513.111}
SPL {X  -150.765, Y  +328.959, Z    +0.000, E1  +313.136, E3 -334529.858}
SPL {X  -148.834, Y  +323.804, Z    +0.000, E1  +313.556, E3 -334541.510}
SPL {X  -147.343, Y  +320.157, Z    +0.000, E1  +313.838, E3 -334549.800}
SPL {X  -142.380, Y  +309.529, Z    +0.000, E1  +319.953, E3 -334622.561}
ENDSPLINE

SPLINE
SPL {X  -153.420, Y  +337.122, Z    +0.000, E1  +333.501, E3 -334680.058}
SPL {X  -157.288, Y  +353.220, Z    +0.000, E1  +341.134, E3 -334692.104}
SPL {X  -159.049, Y  +365.172, Z    +0.000, E1  +347.392, E3 -334697.657}
SPL {X  -159.881, Y  +376.607, Z    +0.000, E1  +353.914, E3 -334700.886}
SPL {X  -159.990, Y  +384.736, Z    +0.000, E1  +359.276, E3 -334702.137}
SPL {X  -159.990, Y  +389.821, Z    +0.000, E1  +363.632, E3 -334702.790}
SPL {X  -159.990, Y  +395.106, Z    +0.000, E1  +369.154, E3 -334703.736}
SPL {X  -159.990, Y  +400.303, Z    +0.000, E1  +374.927, E3 -334705.057}
SPL {X  -159.990, Y  +408.423, Z    +0.000, E1  +383.302, E3 -334708.137}
SPL {X  -159.990, Y  +438.418, Z    +0.000, E1  +401.067, E3 -334729.709}
SPL {X  -159.990, Y  +482.913, Z    +0.000, E1  +407.036, E3 -334789.064}
SPL {X  -159.990, Y  +489.230, Z    +0.000, E1  +407.019, E3 -334801.575}
SPL {X  -159.990, Y  +495.241, Z    +0.000, E1  +407.026, E3 -334813.455}
SPL {X  -159.990, Y  +501.001, Z    +0.000, E1  +407.020, E3 -334824.831}
SPL {X  -159.990, Y  +506.758, Z    +0.000, E1  +407.038, E3 -334836.177}
SPL {X  -159.990, Y  +512.807, Z    +0.000, E1  +407.022, E3 -334848.169}
SPL {X  -159.990, Y  +518.043, Z    +0.000, E1  +407.016, E3 -334858.546}
SPL {X  -159.990, Y  +523.058, Z    +0.000, E1  +407.015, E3 -334868.462}
SPL {X  -159.990, Y  +527.746, Z    +0.000, E1  +407.012, E3 -334877.736}
SPL {X  -159.990, Y  +533.771, Z    +0.000, E1  +407.034, E3 -334889.620}
SPL {X  -159.990, Y  +542.379, Z    +0.000, E1  +407.067, E3 -334906.590}
SPL {X  -159.990, Y  +549.846, Z    +0.000, E1  +407.016, E3 -334921.435}
SPL {X  -159.990, Y  +554.843, Z    +0.000, E1  +407.014, E3 -334931.314}
SPL {X  -159.990, Y  +560.453, Z    +0.000, E1  +407.023, E3 -334942.396}
SPL {X  -159.990, Y  +566.612, Z    +0.000, E1  +407.022, E3 -334954.579}
SPL {X  -159.990, Y  +572.901, Z    +0.000, E1  +407.028, E3 -334966.990}
SPL {X  -159.990, Y  +578.640, Z    +0.000, E1  +407.021, E3 -334978.342}
SPL {X  -159.990, Y  +583.515, Z    +0.000, E1  +407.019, E3 -334987.981}
SPL {X  -159.990, Y  +589.675, Z    +0.000, E1  +407.042, E3 -335000.119}
SPL {X  -159.990, Y  +596.627, Z    +0.000, E1  +407.034, E3 -335013.859}
SPL {X  -159.990, Y  +602.039, Z    +0.000, E1  +407.021, E3 -335024.566}
SPL {X  -159.990, Y  +607.106, Z    +0.000, E1  +407.028, E3 -335034.573}
SPL {X  -159.990, Y  +612.418, Z    +0.000, E1  +407.023, E3 -335045.085}
SPL {X  -159.990, Y  +618.496, Z    +0.000, E1  +407.049, E3 -335057.051}
SPL {X  -159.990, Y  +624.357, Z    +0.000, E1  +407.020, E3 -335068.677}
SPL {X  -159.990, Y  +629.711, Z    +0.000, E1  +407.034, E3 -335079.247}
SPL {X  -159.990, Y  +635.041, Z    +0.000, E1  +407.022, E3 -335089.791}
SPL {X  -159.990, Y  +639.998, Z    +0.000, E1  +407.027, E3 -335099.583}
SPL {X  -159.990, Y  +646.188, Z    +0.000, E1  +407.041, E3 -335111.810}
SPL {X  -159.990, Y  +652.067, Z    +0.000, E1  +407.023, E3 -335123.445}
SPL {X  -159.990, Y  +657.109, Z    +0.000, E1  +407.025, E3 -335133.424}
SPL {X  -159.990, Y  +662.651, Z    +0.000, E1  +407.027, E3 -335144.380}
SPL {X  -159.990, Y  +668.015, Z    +0.000, E1  +407.025, E3 -335154.980}
SPL {X  -159.972, Y  +673.909, Z    +0.000, E1  +407.029, E3 -335166.646}
SPL {X  -159.776, Y  +679.772, Z    +0.000, E1  +406.992, E3 -335178.447}
SPL {X  -159.384, Y  +685.411, Z    +0.000, E1  +406.921, E3 -335190.008}
SPL {X  -158.642, Y  +692.228, Z    +0.000, E1  +406.819, E3 -335204.224}
SPL {X  -157.651, Y  +698.760, Z    +0.000, E1  +406.609, E3 -335218.218}
SPL {X  -156.719, Y  +703.686, Z    +0.000, E1  +406.438, E3 -335228.911}
SPL {X  -155.778, Y  +707.970, Z    +0.000, E1  +406.262, E3 -335238.386}
SPL {X  -154.419, Y  +713.351, Z    +0.000, E1  +406.025, E3 -335250.417}
SPL {X  -152.913, Y  +718.557, Z    +0.000, E1  +405.729, E3 -335262.269}
SPL {X  -151.262, Y  +723.621, Z    +0.000, E1  +405.429, E3 -335273.936}
SPL {X  -149.074, Y  +729.584, Z    +0.000, E1  +405.040, E3 -335287.864}
SPL {X  -142.577, Y  +744.086, Z    +0.000, E1  +400.686, E3 -335354.070}
ENDSPLINE

SPLINE
SPL {X  -152.566, Y  +719.671, Z    +0.000, E1  +387.682, E3 -335424.541}
SPL {X  -158.253, Y  +695.011, Z    +0.000, E1  +375.913, E3 -335441.213}
SPL {X  -159.486, Y  +684.192, Z    +0.000, E1  +369.965, E3 -335445.160}
SPL {X  -159.898, Y  +676.924, Z    +0.000, E1  +365.683, E3 -335446.858}
SPL {X  -159.990, Y  +671.720, Z    +0.000, E1  +362.298, E3 -335447.698}
SPL {X  -159.990, Y  +668.164, Z    +0.000, E1  +359.695, E3 -335448.113}
SPL {X  -159.990, Y  +665.062, Z    +0.000, E1  +356.961, E3 -335448.453}
SPL {X  -159.990, Y  +660.795, Z    +0.000, E1  +352.651, E3 -335449.115}
SPL {X  -159.990, Y  +654.574, Z    +0.000, E1  +345.673, E3 -335450.570}
SPL {X  -159.990, Y  +647.816, Z    +0.000, E1  +338.252, E3 -335452.822}
SPL {X  -159.990, Y  +640.751, Z    +0.000, E1  +331.747, E3 -335456.415}
SPL {X  -159.990, Y  +611.706, Z    +0.000, E1  +317.244, E3 -335479.189}
SPL {X  -159.990, Y  +567.814, Z    +0.000, E1  +312.360, E3 -335539.278}
SPL {X  -159.990, Y  +558.774, Z    +0.000, E1  +312.384, E3 -335556.844}
SPL {X  -159.990, Y  +550.551, Z    +0.000, E1  +312.385, E3 -335572.785}
SPL {X  -159.990, Y  +542.502, Z    +0.000, E1  +312.392, E3 -335588.400}
SPL {X  -159.990, Y  +536.986, Z    +0.000, E1  +312.423, E3 -335599.120}
SPL {X  -159.990, Y  +532.938, Z    +0.000, E1  +312.415, E3 -335606.947}
SPL {X  -159.990, Y  +525.893, Z    +0.000, E1  +312.375, E3 -335620.560}
SPL {X  -159.990, Y  +518.864, Z    +0.000, E1  +312.415, E3 -335634.242}
SPL {X  -159.990, Y  +512.328, Z    +0.000, E1  +312.388, E3 -335646.876}
SPL {X  -159.990, Y  +505.755, Z    +0.000, E1  +312.413, E3 -335659.654}
ENDSPLINE

SPLINE
SPL {X  -159.990, Y  +517.758, Z    +0.000, E1  +318.109, E3 -335667.376}
ENDSPLINE

SPLINE
SPL {X  -159.990, Y  +516.975, Z    +0.000, E1  +319.588, E3 -335678.440}
SPL {X  -159.990, Y  +508.583, Z    +0.000, E1  +318.552, E3 -335692.745}
SPL {X  -159.990, Y  +499.983, Z    +0.000, E1  +317.561, E3 -335707.199}
SPL {X  -159.990, Y  +492.624, Z    +0.000, E1  +316.776, E3 -335719.303}
SPL {X  -159.990, Y  +485.551, Z    +0.000, E1  +316.053, E3 -335730.853}
SPL {X  -159.990, Y  +477.585, Z    +0.000, E1  +315.156, E3 -335742.764}
SPL {X  -159.990, Y  +470.785, Z    +0.000, E1  +314.453, E3 -335752.936}
SPL {X  -159.990, Y  +463.371, Z    +0.000, E1  +313.690, E3 -335763.661}
SPL {X  -159.990, Y  +455.469, Z    +0.000, E1  +312.807, E3 -335774.187}
SPL {X  -159.990, Y  +445.848, Z    +0.000, E1  +311.866, E3 -335787.280}
SPL {X  -159.990, Y  +436.400, Z    +0.000, E1  +311.449, E3 -335802.661}
SPL {X  -159.990, Y  +429.614, Z    +0.000, E1  +311.486, E3 -335815.451}
SPL {X  -159.990, Y  +423.677, Z    +0.000, E1  +311.471, E3 -335826.563}
SPL {X  -159.990, Y  +417.714, Z    +0.000, E1  +311.484, E3 -335837.773}
SPL {X  -159.990, Y  +412.449, Z    +0.000, E1  +311.483, E3 -335847.634}
SPL {X  -159.990, Y  +406.256, Z    +0.000, E1  +311.459, E3 -335859.201}
SPL {X  -159.990, Y  +399.971, Z    +0.000, E1  +311.480, E3 -335871.016}
SPL {X  -159.990, Y  +394.711, Z    +0.000, E1  +311.476, E3 -335880.874}
SPL {X  -159.990, Y  +387.710, Z    +0.000, E1  +311.455, E3 -335893.997}
SPL {X  -159.966, Y  +379.751, Z    +0.000, E1  +311.465, E3 -335908.961}
SPL {X  -159.734, Y  +373.449, Z    +0.000, E1  +311.528, E3 -335921.065}
SPL {X  -159.230, Y  +366.920, Z    +0.000, E1  +311.592, E3 -335933.809}
SPL {X  -158.532, Y  +360.951, Z    +0.000, E1  +311.745, E3 -335945.782}
SPL {X  -157.692, Y  +355.479, Z    +0.000, E1  +311.882, E3 -335956.910}
SPL {X  -156.349, Y  +348.560, Z    +0.000, E1  +312.101, E3 -335971.249}
SPL {X  -154.984, Y  +342.790, Z    +0.000, E1  +312.392, E3 -335983.547}
SPL {X  -153.247, Y  +336.540, Z    +0.000, E1  +312.660, E3 -335996.982}
SPL {X  -150.765, Y  +328.959, Z    +0.000, E1  +313.136, E3 -336013.729}
SPL {X  -148.834, Y  +323.804, Z    +0.000, E1  +313.556, E3 -336025.381}
SPL {X  -147.343, Y  +320.157, Z    +0.000, E1  +313.838, E3 -336033.671}
SPL {X  -142.380, Y  +309.529, Z    +0.000, E1  +319.953, E3 -336106.431}
ENDSPLINE

SPLINE
SPL {X  -153.420, Y  +337.122, Z    +0.000, E1  +333.501, E3 -336163.929}
SPL {X  -157.288, Y  +353.220, Z    +0.000, E1  +341.134, E3 -336175.975}
SPL {X  -159.049, Y  +365.172, Z    +0.000, E1  +347.392, E3 -336181.528}
SPL {X  -159.749, Y  +373.719, Z    +0.000, E1  +352.250, E3 -336184.149}
SPL {X  -159.988, Y  +381.741, Z    +0.000, E1  +357.172, E3 -336185.624}
SPL {X  -159.990, Y  +387.352, Z    +0.000, E1  +361.387, E3 -336186.326}
SPL {X  -159.990, Y  +391.188, Z    +0.000, E1  +365.082, E3 -336186.866}
SPL {X  -159.990, Y  +395.106, Z    +0.000, E1  +369.154, E3 -336187.607}
SPL {X  -159.990, Y  +400.303, Z    +0.000, E1  +374.927, E3 -336188.928}
SPL {X  -159.990, Y  +408.423, Z    +0.000, E1  +383.302, E3 -336192.008}
SPL {X  -159.990, Y  +438.418, Z    +0.000, E1  +401.067, E3 -336213.580}
SPL {X  -159.990, Y  +482.913, Z    +0.000, E1  +407.036, E3 -336272.935}
SPL {X  -159.990, Y  +489.230, Z    +0.000, E1  +407.019, E3 -336285.446}
SPL {X  -159.990, Y  +495.241, Z    +0.000, E1  +407.026, E3 -336297.326}
SPL {X  -159.990, Y  +501.001, Z    +0.000, E1  +407.020, E3 -336308.702}
SPL {X  -159.990, Y  +506.758, Z    +0.000, E1  +407.038, E3 -336320.048}
SPL {X  -159.990, Y  +512.807, Z    +0.000, E1  +407.022, E3 -336332.039}
SPL {X  -159.990, Y  +518.043, Z    +0.000, E1  +407.016, E3 -336342.417}
SPL {X  -159.990, Y  +523.058, Z    +0.000, E1  +407.015, E3 -336352.333}
SPL {X  -159.990, Y  +527.746, Z    +0.000, E1  +407.012, E3 -336361.607}
SPL {X  -159.990, Y  +533.771, Z    +0.000, E1  +407.034, E3 -336373.491}
SPL {X  -159.990, Y  +542.379, Z    +0.000, E1  +407.067, E3 -336390.461}
SPL {X  -159.990, Y  +549.846, Z    +0.000, E1  +407.016, E3 -336405.306}
SPL {X  -159.990, Y  +554.843, Z    +0.000, E1  +407.014, E3 -336415.184}
SPL {X  -159.990, Y  +560.453, Z    +0.000, E1  +407.023, E3 -336426.267}
SPL {X  -159.990, Y  +566.612, Z    +0.000, E1  +407.022, E3 -336438.450}
SPL {X  -159.990, Y  +572.901, Z    +0.000, E1  +407.028, E3 -336450.861}
SPL {X  -159.990, Y  +578.640, Z    +0.000, E1  +407.021, E3 -336462.213}
SPL {X  -159.990, Y  +584.969, Z    +0.000, E1  +407.043, E3 -336474.695}
SPL {X  -159.990, Y  +591.074, Z    +0.000, E1  +407.017, E3 -336486.785}
SPL {X  -159.990, Y  +596.627, Z    +0.000, E1  +407.034, E3 -336497.730}
SPL {X  -159.990, Y  +602.039, Z    +0.000, E1  +407.021, E3 -336508.437}
SPL {X  -159.990, Y  +607.106, Z    +0.000, E1  +407.028, E3 -336518.444}
SPL {X  -159.990, Y  +612.418, Z    +0.000, E1  +407.023, E3 -336528.956}
SPL {X  -159.990, Y  +618.496, Z    +0.000, E1  +407.049, E3 -336540.922}
SPL {X  -159.990, Y  +624.357, Z    +0.000, E1  +407.020, E3 -336552.548}
SPL {X  -159.990, Y  +629.711, Z    +0.000, E1  +407.034, E3 -336563.118}
SPL {X  -159.990, Y  +635.041, Z    +0.000, E1  +407.022, E3 -336573.662}
SPL {X  -159.990, Y  +639.998, Z    +0.000, E1  +407.027, E3 -336583.454}
SPL {X  -159.990, Y  +646.188, Z    +0.000, E1  +407.041, E3 -336595.680}
SPL {X  -159.990, Y  +652.067, Z    +0.000, E1  +407.023, E3 -336607.316}
SPL {X  -159.990, Y  +657.109, Z    +0.000, E1  +407.025, E3 -336617.295}
SPL {X  -159.990, Y  +662.651, Z    +0.000, E1  +407.027, E3 -336628.251}
SPL {X  -159.990, Y  +668.015, Z    +0.000, E1  +407.025, E3 -336638.851}
SPL {X  -159.972, Y  +673.909, Z    +0.000, E1  +407.029, E3 -336650.517}
SPL {X  -159.776, Y  +679.772, Z    +0.000, E1  +406.992, E3 -336662.318}
SPL {X  -159.384, Y  +685.411, Z    +0.000, E1  +406.921, E3 -336673.879}
SPL {X  -158.642, Y  +692.228, Z    +0.000, E1  +406.819, E3 -336688.094}
SPL {X  -157.651, Y  +698.760, Z    +0.000, E1  +406.609, E3 -336702.089}
SPL {X  -156.719, Y  +703.686, Z    +0.000, E1  +406.438, E3 -336712.782}
SPL {X  -155.778, Y  +707.970, Z    +0.000, E1  +406.262, E3 -336722.257}
SPL {X  -154.419, Y  +713.351, Z    +0.000, E1  +406.025, E3 -336734.288}
SPL {X  -152.913, Y  +718.557, Z    +0.000, E1  +405.729, E3 -336746.140}
SPL {X  -151.262, Y  +723.621, Z    +0.000, E1  +405.429, E3 -336757.807}
SPL {X  -149.074, Y  +729.584, Z    +0.000, E1  +405.040, E3 -336771.735}
SPL {X  -142.577, Y  +744.086, Z    +0.000, E1  +400.686, E3 -336837.941}
ENDSPLINE

SPLINE
SPL {X  -152.566, Y  +719.671, Z    +0.000, E1  +387.682, E3 -336908.412}
SPL {X  -158.253, Y  +695.011, Z    +0.000, E1  +375.913, E3 -336925.084}
SPL {X  -159.486, Y  +684.192, Z    +0.000, E1  +369.965, E3 -336929.031}
SPL {X  -159.898, Y  +676.924, Z    +0.000, E1  +365.683, E3 -336930.729}
SPL {X  -159.990, Y  +671.720, Z    +0.000, E1  +362.298, E3 -336931.569}
SPL {X  -159.990, Y  +668.164, Z    +0.000, E1  +359.695, E3 -336931.984}
SPL {X  -159.990, Y  +665.062, Z    +0.000, E1  +356.961, E3 -336932.324}
SPL {X  -159.990, Y  +660.795, Z    +0.000, E1  +352.651, E3 -336932.986}
SPL {X  -159.990, Y  +654.574, Z    +0.000, E1  +345.673, E3 -336934.441}
SPL {X  -159.990, Y  +644.002, Z    +0.000, E1  +334.724, E3 -336938.638}
SPL {X  -159.990, Y  +611.706, Z    +0.000, E1  +317.244, E3 -336963.060}
SPL {X  -159.990, Y  +571.318, Z    +0.000, E1  +312.417, E3 -337016.443}
SPL {X  -159.990, Y  +566.024, Z    +0.000, E1  +312.406, E3 -337026.693}
SPL {X  -159.990, Y  +558.774, Z    +0.000, E1  +312.384, E3 -337040.715}
SPL {X  -159.990, Y  +550.551, Z    +0.000, E1  +312.385, E3 -337056.656}
SPL {X  -159.990, Y  +542.502, Z    +0.000, E1  +312.392, E3 -337072.271}
SPL {X  -159.990, Y  +534.538, Z    +0.000, E1  +312.385, E3 -337087.675}
SPL {X  -159.990, Y  +527.222, Z    +0.000, E1  +312.401, E3 -337101.883}
SPL {X  -159.990, Y  +520.237, Z    +0.000, E1  +312.390, E3 -337115.414}
SPL {X  -159.990, Y  +512.328, Z    +0.000, E1  +312.388, E3 -337130.747}
SPL {X  -159.990, Y  +505.755, Z    +0.000, E1  +312.413, E3 -337143.525}
ENDSPLINE

SPLINE
SPL {X  -159.990, Y  +517.758, Z    +0.000, E1  +318.109, E3 -337151.247}
ENDSPLINE

SPLINE
SPL {X  -159.990, Y  +516.975, Z    +0.000, E1  +319.588, E3 -337162.311}
SPL {X  -159.990, Y  +508.583, Z    +0.000, E1  +318.552, E3 -337176.616}
SPL {X  -159.990, Y  +502.438, Z    +0.000, E1  +317.876, E3 -337187.119}
SPL {X  -159.990, Y  +494.810, Z    +0.000, E1  +316.979, E3 -337199.535}
SPL {X  -159.990, Y  +487.314, Z    +0.000, E1  +316.246, E3 -337211.903}
SPL {X  -159.990, Y  +479.678, Z    +0.000, E1  +315.383, E3 -337223.574}
SPL {X  -159.990, Y  +470.785, Z    +0.000, E1  +314.453, E3 -337236.807}
SPL {X  -159.990, Y  +463.371, Z    +0.000, E1  +313.690, E3 -337247.532}
SPL {X  -159.990, Y  +455.469, Z    +0.000, E1  +312.807, E3 -337258.058}
SPL {X  -159.990, Y  +449.689, Z    +0.000, E1  +312.264, E3 -337266.048}
SPL {X  -159.990, Y  +441.904, Z    +0.000, E1  +311.574, E3 -337276.885}
SPL {X  -159.990, Y  +434.881, Z    +0.000, E1  +311.481, E3 -337289.433}
SPL {X  -159.990, Y  +427.340, Z    +0.000, E1  +311.445, E3 -337303.527}
SPL {X  -159.990, Y  +418.926, Z    +0.000, E1  +311.461, E3 -337319.336}
SPL {X  -159.990, Y  +412.449, Z    +0.000, E1  +311.483, E3 -337331.504}
SPL {X  -159.990, Y  +406.256, Z    +0.000, E1  +311.459, E3 -337343.072}
SPL {X  -159.990, Y  +399.971, Z    +0.000, E1  +311.480, E3 -337354.887}
SPL {X  -159.990, Y  +392.623, Z    +0.000, E1  +311.440, E3 -337368.617}
SPL {X  -159.990, Y  +385.787, Z    +0.000, E1  +311.488, E3 -337381.525}
SPL {X  -159.966, Y  +379.751, Z    +0.000, E1  +311.465, E3 -337392.832}
SPL {X  -159.734, Y  +373.449, Z    +0.000, E1  +311.528, E3 -337404.936}
SPL {X  -159.230, Y  +366.920, Z    +0.000, E1  +311.592, E3 -337417.680}
SPL {X  -158.532, Y  +360.951, Z    +0.000, E1  +311.745, E3 -337429.653}
SPL {X  -157.692, Y  +355.479, Z    +0.000, E1  +311.882, E3 -337440.781}
SPL {X  -156.349, Y  +348.560, Z    +0.000, E1  +312.101, E3 -337455.120}
SPL {X  -154.984, Y  +342.790, Z    +0.000, E1  +312.392, E3 -337467.418}
SPL {X  -153.247, Y  +336.540, Z    +0.000, E1  +312.660, E3 -337480.853}
SPL {X  -150.765, Y  +328.959, Z    +0.000, E1  +313.136, E3 -337497.599}
SPL {X  -148.834, Y  +323.804, Z    +0.000, E1  +313.556, E3 -337509.252}
SPL {X  -147.343, Y  +320.157, Z    +0.000, E1  +313.838, E3 -337517.542}
SPL {X  -142.380, Y  +309.529, Z    +0.000, E1  +319.953, E3 -337590.302}
ENDSPLINE

SPLINE
SPL {X  -153.420, Y  +337.122, Z    +0.000, E1  +333.501, E3 -337647.800}
SPL {X  -157.288, Y  +353.220, Z    +0.000, E1  +341.134, E3 -337659.846}
SPL {X  -159.049, Y  +365.172, Z    +0.000, E1  +347.392, E3 -337665.399}
SPL {X  -159.749, Y  +373.719, Z    +0.000, E1  +352.250, E3 -337668.020}
SPL {X  -159.988, Y  +381.741, Z    +0.000, E1  +357.172, E3 -337669.495}
SPL {X  -159.990, Y  +387.352, Z    +0.000, E1  +361.387, E3 -337670.197}
SPL {X  -159.990, Y  +391.188, Z    +0.000, E1  +365.082, E3 -337670.737}
SPL {X  -159.990, Y  +395.106, Z    +0.000, E1  +369.154, E3 -337671.478}
SPL {X  -159.990, Y  +400.303, Z    +0.000, E1  +374.927, E3 -337672.799}
SPL {X  -159.990, Y  +408.423, Z    +0.000, E1  +383.302, E3 -337675.879}
SPL {X  -159.990, Y  +438.418, Z    +0.000, E1  +401.067, E3 -337697.451}
SPL {X  -159.990, Y  +482.913, Z    +0.000, E1  +407.036, E3 -337756.806}
SPL {X  -159.990, Y  +489.230, Z    +0.000, E1  +407.019, E3 -337769.317}
SPL {X  -159.990, Y  +495.241, Z    +0.000, E1  +407.026, E3 -337781.196}
SPL {X  -159.990, Y  +501.001, Z    +0.000, E1  +407.020, E3 -337792.573}
SPL {X  -159.990, Y  +506.758, Z    +0.000, E1  +407.038, E3 -337803.919}
SPL {X  -159.990, Y  +512.807, Z    +0.000, E1  +407.022, E3 -337815.910}
SPL {X  -159.990, Y  +518.043, Z    +0.000, E1  +407.016, E3 -337826.288}
SPL {X  -159.990, Y  +523.058, Z    +0.000, E1  +407.015, E3 -337836.204}
SPL {X  -159.990, Y  +527.746, Z    +0.000, E1  +407.012, E3 -337845.478}
SPL {X  -159.990, Y  +533.771, Z    +0.000, E1  +407.034, E3 -337857.362}
SPL {X  -159.990, Y  +542.379, Z    +0.000, E1  +407.067, E3 -337874.332}
SPL {X  -159.990, Y  +549.846, Z    +0.000, E1  +407.016, E3 -337889.177}
SPL {X  -159.990, Y  +554.843, Z    +0.000, E1  +407.014, E3 -337899.055}
SPL {X  -159.990, Y  +560.453, Z    +0.000, E1  +407.023, E3 -337910.138}
SPL {X  -159.990, Y  +566.612, Z    +0.000, E1  +407.022, E3 -337922.321}
SPL {X  -159.990, Y  +572.901, Z    +0.000, E1  +407.028, E3 -337934.732}
SPL {X  -159.990, Y  +578.640, Z    +0.000, E1  +407.021, E3 -337946.084}
SPL {X  -159.990, Y  +583.515, Z    +0.000, E1  +407.019, E3 -337955.723}
SPL {X  -159.990, Y  +589.675, Z    +0.000, E1  +407.042, E3 -337967.861}
SPL {X  -159.990, Y  +596.627, Z    +0.000, E1  +407.034, E3 -337981.601}
SPL {X  -159.990, Y  +602.039, Z    +0.000, E1  +407.021, E3 -337992.308}
SPL {X  -159.990, Y  +607.106, Z    +0.000, E1  +407.028, E3 -338002.315}
SPL {X  -159.990, Y  +612.418, Z    +0.000, E1  +407.023, E3 -338012.827}
SPL {X  -159.990, Y  +618.496, Z    +0.000, E1  +407.049, E3 -338024.793}
SPL {X  -159.990, Y  +624.357, Z    +0.000, E1  +407.020, E3 -338036.419}
SPL {X  -159.990, Y  +629.711, Z    +0.000, E1  +407.034, E3 -338046.989}
SPL {X  -159.990, Y  +635.041, Z    +0.000, E1  +407.022, E3 -338057.533}
SPL {X  -159.990, Y  +639.998, Z    +0.000, E1  +407.027, E3 -338067.325}
SPL {X  -159.990, Y  +646.188, Z    +0.000, E1  +407.041, E3 -338079.551}
SPL {X  -159.990, Y  +652.067, Z    +0.000, E1  +407.023, E3 -338091.187}
SPL {X  -159.990, Y  +657.109, Z    +0.000, E1  +407.025, E3 -338101.166}
SPL {X  -159.990, Y  +662.651, Z    +0.000, E1  +407.027, E3 -338112.122}
SPL {X  -159.990, Y  +668.015, Z    +0.000, E1  +407.025, E3 -338122.722}
SPL {X  -159.972, Y  +673.909, Z    +0.000, E1  +407.029, E3 -338134.388}
SPL {X  -159.776, Y  +679.772, Z    +0.000, E1  +406.992, E3 -338146.189}
SPL {X  -159.384, Y  +685.411, Z    +0.000, E1  +406.921, E3 -338157.750}
SPL {X  -158.839, Y  +690.657, Z    +0.000, E1  +406.819, E3 -338168.704}
SPL {X  -157.875, Y  +697.431, Z    +0.000, E1  +406.688, E3 -338183.044}
SPL {X  -156.719, Y  +703.686, Z    +0.000, E1  +406.438, E3 -338196.653}
SPL {X  -155.778, Y  +707.970, Z    +0.000, E1  +406.262, E3 -338206.128}
SPL {X  -154.419, Y  +713.351, Z    +0.000, E1  +406.025, E3 -338218.159}
SPL {X  -152.913, Y  +718.557, Z    +0.000, E1  +405.729, E3 -338230.011}
SPL {X  -151.262, Y  +723.621, Z    +0.000, E1  +405.429, E3 -338241.678}
SPL {X  -149.074, Y  +729.584, Z    +0.000, E1  +405.040, E3 -338255.606}
SPL {X  -142.577, Y  +744.086, Z    +0.000, E1  +400.686, E3 -338321.812}
ENDSPLINE

SPLINE
SPL {X  -152.566, Y  +719.671, Z    +0.000, E1  +387.682, E3 -338392.283}
SPL {X  -158.253, Y  +695.011, Z    +0.000, E1  +375.913, E3 -338408.955}
SPL {X  -159.486, Y  +684.192, Z    +0.000, E1  +369.965, E3 -338412.902}
SPL {X  -159.898, Y  +676.924, Z    +0.000, E1  +365.683, E3 -338414.599}
SPL {X  -159.990, Y  +671.720, Z    +0.000, E1  +362.298, E3 -338415.440}
SPL {X  -159.990, Y  +668.164, Z    +0.000, E1  +359.695, E3 -338415.855}
SPL {X  -159.990, Y  +665.062, Z    +0.000, E1  +356.961, E3 -338416.195}
SPL {X  -159.990, Y  +660.795, Z    +0.000, E1  +352.651, E3 -338416.857}
SPL {X  -159.990, Y  +654.574, Z    +0.000, E1  +345.673, E3 -338418.312}
SPL {X  -159.990, Y  +647.816, Z    +0.000, E1  +338.252, E3 -338420.563}
SPL {X  -159.990, Y  +640.751, Z    +0.000, E1  +331.747, E3 -338424.157}
SPL {X  -159.990, Y  +611.706, Z    +0.000, E1  +317.244, E3 -338446.931}
SPL {X  -159.990, Y  +567.814, Z    +0.000, E1  +312.360, E3 -338507.020}
SPL {X  -159.990, Y  +558.774, Z    +0.000, E1  +312.384, E3 -338524.586}
SPL {X  -159.990, Y  +550.551, Z    +0.000, E1  +312.385, E3 -338540.527}
SPL {X  -159.990, Y  +542.502, Z    +0.000, E1  +312.392, E3 -338556.142}
SPL {X  -159.990, Y  +536.986, Z    +0.000, E1  +312.423, E3 -338566.862}
SPL {X  -159.990, Y  +532.938, Z    +0.000, E1  +312.415, E3 -338574.689}
SPL {X  -159.990, Y  +525.893, Z    +0.000, E1  +312.375, E3 -338588.302}
SPL {X  -159.990, Y  +518.864, Z    +0.000, E1  +312.415, E3 -338601.984}
SPL {X  -159.990, Y  +512.328, Z    +0.000, E1  +312.388, E3 -338614.618}
SPL {X  -159.990, Y  +505.755, Z    +0.000, E1  +312.413, E3 -338627.395}
ENDSPLINE

SPLINE
SPL {X  -159.990, Y  +517.758, Z    +0.000, E1  +318.109, E3 -338635.118}
ENDSPLINE

SPLINE
SPL {X  -159.990, Y  +516.975, Z    +0.000, E1  +319.588, E3 -338646.182}
SPL {X  -159.990, Y  +508.583, Z    +0.000, E1  +318.552, E3 -338660.487}
SPL {X  -159.990, Y  +499.983, Z    +0.000, E1  +317.561, E3 -338674.941}
SPL {X  -159.990, Y  +492.624, Z    +0.000, E1  +316.776, E3 -338687.045}
SPL {X  -159.990, Y  +485.551, Z    +0.000, E1  +316.053, E3 -338698.595}
SPL {X  -159.990, Y  +477.585, Z    +0.000, E1  +315.156, E3 -338710.506}
SPL {X  -159.990, Y  +470.785, Z    +0.000, E1  +314.453, E3 -338720.678}
SPL {X  -159.990, Y  +463.371, Z    +0.000, E1  +313.690, E3 -338731.403}
SPL {X  -159.990, Y  +455.469, Z    +0.000, E1  +312.807, E3 -338741.929}
SPL {X  -159.990, Y  +445.848, Z    +0.000, E1  +311.866, E3 -338755.022}
SPL {X  -159.990, Y  +436.400, Z    +0.000, E1  +311.449, E3 -338770.403}
SPL {X  -159.990, Y  +429.614, Z    +0.000, E1  +311.486, E3 -338783.193}
SPL {X  -159.990, Y  +423.677, Z    +0.000, E1  +311.471, E3 -338794.305}
SPL {X  -159.990, Y  +417.714, Z    +0.000, E1  +311.484, E3 -338805.515}
SPL {X  -159.990, Y  +412.449, Z    +0.000, E1  +311.483, E3 -338815.375}
SPL {X  -159.990, Y  +406.256, Z    +0.000, E1  +311.459, E3 -338826.943}
SPL {X  -159.990, Y  +399.971, Z    +0.000, E1  +311.480, E3 -338838.758}
SPL {X  -159.990, Y  +394.711, Z    +0.000, E1  +311.476, E3 -338848.616}
SPL {X  -159.990, Y  +387.710, Z    +0.000, E1  +311.455, E3 -338861.739}
SPL {X  -159.966, Y  +379.751, Z    +0.000, E1  +311.465, E3 -338876.703}
SPL {X  -159.734, Y  +373.449, Z    +0.000, E1  +311.528, E3 -338888.807}
SPL {X  -159.230, Y  +366.920, Z    +0.000, E1  +311.592, E3 -338901.551}
SPL {X  -158.532, Y  +360.951, Z    +0.000, E1  +311.745, E3 -338913.524}
SPL {X  -157.692, Y  +355.479, Z    +0.000, E1  +311.882, E3 -338924.652}
SPL {X  -156.349, Y  +348.560, Z    +0.000, E1  +312.101, E3 -338938.991}
SPL {X  -154.984, Y  +342.790, Z    +0.000, E1  +312.392, E3 -338951.289}
SPL {X  -153.247, Y  +336.540, Z    +0.000, E1  +312.660, E3 -338964.724}
SPL {X  -150.765, Y  +328.959, Z    +0.000, E1  +313.136, E3 -338981.470}
SPL {X  -148.834, Y  +323.804, Z    +0.000, E1  +313.556, E3 -338993.123}
SPL {X  -147.343, Y  +320.157, Z    +0.000, E1  +313.838, E3 -339001.413}
SPL {X  -142.380, Y  +309.529, Z    +0.000, E1  +319.953, E3 -339074.173}
ENDSPLINE

SPLINE
SPL {X  -153.420, Y  +337.122, Z    +0.000, E1  +333.501, E3 -339131.671}
SPL {X  -157.288, Y  +353.220, Z    +0.000, E1  +341.134, E3 -339143.717}
SPL {X  -159.049, Y  +365.172, Z    +0.000, E1  +347.392, E3 -339149.270}
SPL {X  -159.749, Y  +373.719, Z    +0.000, E1  +352.250, E3 -339151.890}
SPL {X  -159.988, Y  +381.741, Z    +0.000, E1  +357.172, E3 -339153.366}
SPL {X  -159.990, Y  +387.352, Z    +0.000, E1  +361.387, E3 -339154.068}
SPL {X  -159.990, Y  +391.188, Z    +0.000, E1  +365.082, E3 -339154.608}
SPL {X  -159.990, Y  +395.106, Z    +0.000, E1  +369.154, E3 -339155.349}
SPL {X  -159.990, Y  +400.303, Z    +0.000, E1  +374.927, E3 -339156.670}
SPL {X  -159.990, Y  +408.423, Z    +0.000, E1  +383.302, E3 -339159.750}
SPL {X  -159.990, Y  +438.418, Z    +0.000, E1  +401.067, E3 -339181.322}
SPL {X  -159.990, Y  +482.913, Z    +0.000, E1  +407.036, E3 -339240.677}
SPL {X  -159.990, Y  +489.230, Z    +0.000, E1  +407.019, E3 -339253.188}
SPL {X  -159.990, Y  +495.241, Z    +0.000, E1  +407.026, E3 -339265.067}
SPL {X  -159.990, Y  +501.001, Z    +0.000, E1  +407.020, E3 -339276.444}
SPL {X  -159.990, Y  +506.758, Z    +0.000, E1  +407.038, E3 -339287.790}
SPL {X  -159.990, Y  +512.807, Z    +0.000, E1  +407.022, E3 -339299.781}
SPL {X  -159.990, Y  +518.043, Z    +0.000, E1  +407.016, E3 -339310.159}
SPL {X  -159.990, Y  +523.058, Z    +0.000, E1  +407.015, E3 -339320.075}
SPL {X  -159.990, Y  +527.746, Z    +0.000, E1  +407.012, E3 -339329.349}
SPL {X  -159.990, Y  +533.771, Z    +0.000, E1  +407.034, E3 -339341.233}
SPL {X  -159.990, Y  +542.379, Z    +0.000, E1  +407.067, E3 -339358.203}
SPL {X  -159.990, Y  +549.846, Z    +0.000, E1  +407.016, E3 -339373.048}
SPL {X  -159.990, Y  +554.843, Z    +0.000, E1  +407.014, E3 -339382.926}
SPL {X  -159.990, Y  +560.453, Z    +0.000, E1  +407.023, E3 -339394.009}
SPL {X  -159.990, Y  +566.612, Z    +0.000, E1  +407.022, E3 -339406.192}
SPL {X  -159.990, Y  +572.901, Z    +0.000, E1  +407.028, E3 -339418.603}
SPL {X  -159.990, Y  +578.640, Z    +0.000, E1  +407.021, E3 -339429.955}
SPL {X  -159.990, Y  +583.515, Z    +0.000, E1  +407.019, E3 -339439.594}
SPL {X  -159.990, Y  +589.675, Z    +0.000, E1  +407.042, E3 -339451.732}
SPL {X  -159.990, Y  +596.627, Z    +0.000, E1  +407.034, E3 -339465.472}
SPL {X  -159.990, Y  +602.039, Z    +0.000, E1  +407.021, E3 -339476.179}
SPL {X  -159.990, Y  +607.106, Z    +0.000, E1  +407.028, E3 -339486.186}
SPL {X  -159.990, Y  +612.418, Z    +0.000, E1  +407.023, E3 -339496.698}
SPL {X  -159.990, Y  +618.496, Z    +0.000, E1  +407.049, E3 -339508.664}
SPL {X  -159.990, Y  +624.357, Z    +0.000, E1  +407.020, E3 -339520.290}
SPL {X  -159.990, Y  +629.711, Z    +0.000, E1  +407.034, E3 -339530.859}
SPL {X  -159.990, Y  +635.041, Z    +0.000, E1  +407.022, E3 -339541.404}
SPL {X  -159.990, Y  +639.998, Z    +0.000, E1  +407.027, E3 -339551.196}
SPL {X  -159.990, Y  +646.188, Z    +0.000, E1  +407.041, E3 -339563.422}
SPL {X  -159.990, Y  +652.067, Z    +0.000, E1  +407.023, E3 -339575.058}
SPL {X  -159.990, Y  +657.109, Z    +0.000, E1  +407.025, E3 -339585.037}
SPL {X  -159.990, Y  +662.651, Z    +0.000, E1  +407.027, E3 -339595.993}
SPL {X  -159.990, Y  +668.015, Z    +0.000, E1  +407.025, E3 -339606.593}
SPL {X  -159.972, Y  +673.909, Z    +0.000, E1  +407.029, E3 -339618.259}
SPL {X  -159.776, Y  +679.772, Z    +0.000, E1  +406.992, E3 -339630.060}
SPL {X  -159.384, Y  +685.411, Z    +0.000, E1  +406.921, E3 -339641.621}
SPL {X  -158.839, Y  +690.657, Z    +0.000, E1  +406.819, E3 -339652.575}
SPL {X  -157.875, Y  +697.431, Z    +0.000, E1  +406.688, E3 -339666.915}
SPL {X  -156.719, Y  +703.686, Z    +0.000, E1  +406.438, E3 -339680.524}
SPL {X  -155.778, Y  +707.970, Z    +0.000, E1  +406.262, E3 -339689.999}
SPL {X  -154.419, Y  +713.351, Z    +0.000, E1  +406.025, E3 -339702.030}
SPL {X  -152.913, Y  +718.557, Z    +0.000, E1  +405.729, E3 -339713.882}
SPL {X  -151.262, Y  +723.621, Z    +0.000, E1  +405.429, E3 -339725.548}
SPL {X  -149.074, Y  +729.584, Z    +0.000, E1  +405.040, E3 -339739.477}
SPL {X  -142.577, Y  +744.086, Z    +0.000, E1  +400.686, E3 -339805.683}
ENDSPLINE

SPLINE
SPL {X  -152.566, Y  +719.671, Z    +0.000, E1  +387.682, E3 -339876.154}
SPL {X  -158.253, Y  +695.011, Z    +0.000, E1  +375.913, E3 -339892.826}
SPL {X  -159.486, Y  +684.192, Z    +0.000, E1  +369.965, E3 -339896.772}
SPL {X  -159.898, Y  +676.924, Z    +0.000, E1  +365.683, E3 -339898.470}
SPL {X  -159.990, Y  +671.720, Z    +0.000, E1  +362.298, E3 -339899.311}
SPL {X  -159.990, Y  +668.164, Z    +0.000, E1  +359.695, E3 -339899.726}
SPL {X  -159.990, Y  +665.062, Z    +0.000, E1  +356.961, E3 -339900.066}
SPL {X  -159.990, Y  +660.795, Z    +0.000, E1  +352.651, E3 -339900.728}
SPL {X  -159.990, Y  +654.574, Z    +0.000, E1  +345.673, E3 -339902.183}
SPL {X  -159.990, Y  +647.816, Z    +0.000, E1  +338.252, E3 -339904.434}
SPL {X  -159.990, Y  +640.751, Z    +0.000, E1  +331.747, E3 -339908.028}
SPL {X  -159.990, Y  +611.706, Z    +0.000, E1  +317.244, E3 -339930.802}
SPL {X  -159.990, Y  +567.814, Z    +0.000, E1  +312.360, E3 -339990.891}
SPL {X  -159.990, Y  +558.774, Z    +0.000, E1  +312.384, E3 -340008.457}
SPL {X  -159.990, Y  +550.551, Z    +0.000, E1  +312.385, E3 -340024.398}
SPL {X  -159.990, Y  +542.502, Z    +0.000, E1  +312.392, E3 -340040.013}
SPL {X  -159.990, Y  +536.986, Z    +0.000, E1  +312.423, E3 -340050.733}
SPL {X  -159.990, Y  +532.938, Z    +0.000, E1  +312.415, E3 -340058.560}
SPL {X  -159.990, Y  +525.893, Z    +0.000, E1  +312.375, E3 -340072.173}
SPL {X  -159.990, Y  +518.864, Z    +0.000, E1  +312.415, E3 -340085.855}
SPL {X  -159.990, Y  +512.328, Z    +0.000, E1  +312.388, E3 -340098.489}
SPL {X  -159.990, Y  +505.755, Z    +0.000, E1  +312.413, E3 -340111.266}
ENDSPLINE

SPLINE
SPL {X  -159.990, Y  +517.758, Z    +0.000, E1  +318.109, E3 -340118.989}
ENDSPLINE

SPLINE
SPL {X  -159.990, Y  +516.975, Z    +0.000, E1  +319.588, E3 -340130.053}
SPL {X  -159.990, Y  +508.583, Z    +0.000, E1  +318.552, E3 -340144.358}
SPL {X  -159.990, Y  +499.983, Z    +0.000, E1  +317.561, E3 -340158.812}
SPL {X  -159.990, Y  +492.624, Z    +0.000, E1  +316.776, E3 -340170.916}
SPL {X  -159.990, Y  +485.551, Z    +0.000, E1  +316.053, E3 -340182.466}
SPL {X  -159.990, Y  +477.585, Z    +0.000, E1  +315.156, E3 -340194.377}
SPL {X  -159.990, Y  +470.785, Z    +0.000, E1  +314.453, E3 -340204.549}
SPL {X  -159.990, Y  +463.371, Z    +0.000, E1  +313.690, E3 -340215.274}
SPL {X  -159.990, Y  +455.469, Z    +0.000, E1  +312.807, E3 -340225.800}
SPL {X  -159.990, Y  +445.848, Z    +0.000, E1  +311.866, E3 -340238.893}
SPL {X  -159.990, Y  +436.400, Z    +0.000, E1  +311.449, E3 -340254.274}
SPL {X  -159.990, Y  +429.614, Z    +0.000, E1  +311.486, E3 -340267.064}
SPL {X  -159.990, Y  +423.677, Z    +0.000, E1  +311.471, E3 -340278.176}
SPL {X  -159.990, Y  +417.714, Z    +0.000, E1  +311.484, E3 -340289.386}
SPL {X  -159.990, Y  +412.449, Z    +0.000, E1  +311.483, E3 -340299.246}
SPL {X  -159.990, Y  +406.256, Z    +0.000, E1  +311.459, E3 -340310.814}
SPL {X  -159.990, Y  +399.971, Z    +0.000, E1  +311.480, E3 -340322.629}
SPL {X  -159.990, Y  +394.711, Z    +0.000, E1  +311.476, E3 -340332.487}
SPL {X  -159.990, Y  +387.710, Z    +0.000, E1  +311.455, E3 -340345.610}
SPL {X  -159.966, Y  +379.751, Z    +0.000, E1  +311.465, E3 -340360.574}
SPL {X  -159.734, Y  +373.449, Z    +0.000, E1  +311.528, E3 -340372.678}
SPL {X  -159.230, Y  +366.920, Z    +0.000, E1  +311.592, E3 -340385.422}
SPL {X  -158.532, Y  +360.951, Z    +0.000, E1  +311.745, E3 -340397.395}
SPL {X  -157.692, Y  +355.479, Z    +0.000, E1  +311.882, E3 -340408.523}
SPL {X  -156.349, Y  +348.560, Z    +0.000, E1  +312.101, E3 -340422.862}
SPL {X  -154.984, Y  +342.790, Z    +0.000, E1  +312.392, E3 -340435.159}
SPL {X  -153.247, Y  +336.540, Z    +0.000, E1  +312.660, E3 -340448.595}
SPL {X  -150.765, Y  +328.959, Z    +0.000, E1  +313.136, E3 -340465.341}
SPL {X  -148.834, Y  +323.804, Z    +0.000, E1  +313.556, E3 -340476.994}
SPL {X  -147.343, Y  +320.157, Z    +0.000, E1  +313.838, E3 -340485.284}
SPL {X  -142.380, Y  +309.529, Z    +0.000, E1  +319.953, E3 -340558.044}
ENDSPLINE

